LIN {X 0,Y 573.461,Z 507.991,A -85,B 0,C 180,E1 -2261.308,E2 -2261.308} C_VEL
LIN {X 0,Y 573.62,Z 497.143,A -85,B 0,C 180,E1 -2262.201,E2 -2262.201} C_VEL
LIN {X 0,Y 573.738,Z 485.26,A -85,B 0,C 180,E1 -2263.008,E2 -2263.008} C_VEL
LIN {X 0,Y 573.946,Z 472.1,A -85,B 0,C 180,E1 -2263.724,E2 -2263.724} C_VEL
LIN {X 0,Y 574.081,Z 458.765,A -85,B 0,C 180,E1 -2264.286,E2 -2264.286} C_VEL
LIN {X 0,Y 574.199,Z 444.491,A -85,B 0,C 180,E1 -2264.728,E2 -2264.728} C_VEL
LIN {X 0,Y 574.308,Z 429.641,A -85,B 0,C 180,E1 -2265.027,E2 -2265.027} C_VEL
LIN {X 0,Y 574.551,Z 299.634,A -85,B 0,C 180,E1 -2266.683,E2 -2266.683} C_VEL
LIN {X 0,Y 573.723,Z 294.688,A -85,B 0,C 180,E1 -2266.799,E2 -2266.799} C_VEL
LIN {X 0,Y 573.965,Z 271.516,A -85,B 0,C 180,E1 -2269.466,E2 -2269.466} C_VEL
LIN {X 0,Y 574.336,Z 247.477,A -85,B 0,C 180,E1 -2272.292,E2 -2272.292} C_VEL
LIN {X 0,Y 574.248,Z 241.135,A -85,B 0,C 180,E1 -2273.056,E2 -2273.056} C_VEL
LIN {X 0,Y 573.273,Z 236.765,A -85,B 0,C 180,E1 -2273.667,E2 -2273.667} C_VEL
LIN {X 0,Y 573.237,Z 236.705,A -85,B 0,C 180,E1 -2276.492,E2 -2276.492} C_VEL
LIN {X 0,Y 573.238,Z 236.705,A -85,B 0,C 180,E1 -2278.564,E2 -2278.564} C_VEL
LIN {X 0,Y 573.224,Z 236.702,A -85,B 0,C 180,E1 -2280.993,E2 -2280.993} C_VEL
LIN {X 0,Y 573.261,Z 236.697,A -85,B 0,C 180,E1 -2283.524,E2 -2283.524} C_VEL
LIN {X 0,Y 573.212,Z 236.706,A -85,B 0,C 180,E1 -2286.051,E2 -2286.051} C_VEL
LIN {X 0,Y 573.239,Z 236.705,A -85,B 0,C 180,E1 -2288.701,E2 -2288.701} C_VEL
LIN {X 0,Y 573.25,Z 236.698,A -85,B 0,C 180,E1 -2291.595,E2 -2291.595} C_VEL
LIN {X 0,Y 573.236,Z 236.707,A -85,B 0,C 180,E1 -2294.332,E2 -2294.332} C_VEL
LIN {X 0,Y 573.236,Z 236.7,A -85,B 0,C 180,E1 -2297.358,E2 -2297.358} C_VEL
LIN {X 0,Y 573.244,Z 236.706,A -85,B 0,C 180,E1 -2300.393,E2 -2300.393} C_VEL
LIN {X 0,Y 573.252,Z 236.696,A -85,B 0,C 180,E1 -2303.078,E2 -2303.078} C_VEL
LIN {X 0,Y 573.268,Z 236.698,A -85,B 0,C 180,E1 -2305.671,E2 -2305.671} C_VEL
LIN {X 0,Y 573.243,Z 236.705,A -85,B 0,C 180,E1 -2308.185,E2 -2308.185} C_VEL
LIN {X 0,Y 573.263,Z 236.695,A -85,B 0,C 180,E1 -2310.634,E2 -2310.634} C_VEL
LIN {X 0,Y 573.248,Z 236.698,A -85,B 0,C 180,E1 -2313.024,E2 -2313.024} C_VEL
LIN {X 0,Y 573.269,Z 236.697,A -85,B 0,C 180,E1 -2315.366,E2 -2315.366} C_VEL
LIN {X 0,Y 573.223,Z 236.703,A -85,B 0,C 180,E1 -2318.419,E2 -2318.419} C_VEL
LIN {X 0,Y 573.271,Z 236.695,A -85,B 0,C 180,E1 -2320.728,E2 -2320.728} C_VEL
LIN {X 0,Y 573.253,Z 236.704,A -85,B 0,C 180,E1 -2323.622,E2 -2323.622} C_VEL
LIN {X 0,Y 573.232,Z 236.7,A -85,B 0,C 180,E1 -2326.53,E2 -2326.53} C_VEL
LIN {X 0,Y 573.255,Z 236.696,A -85,B 0,C 180,E1 -2328.745,E2 -2328.745} C_VEL
LIN {X 0,Y 573.284,Z 236.701,A -85,B 0,C 180,E1 -2331.541,E2 -2331.541} C_VEL
LIN {X 0,Y 573.287,Z 236.694,A -85,B 0,C 180,E1 -2334.372,E2 -2334.372} C_VEL
LIN {X 0,Y 573.302,Z 236.696,A -85,B 0,C 180,E1 -2337.893,E2 -2337.893} C_VEL
LIN {X 0,Y 573.328,Z 236.688,A -85,B 0,C 180,E1 -2340.703,E2 -2340.703} C_VEL
LIN {X 0,Y 573.234,Z 236.71,A -85,B 0,C 180,E1 -2343.515,E2 -2343.515} C_VEL
LIN {X 0,Y 573.286,Z 236.7,A -85,B 0,C 180,E1 -2345.628,E2 -2345.628} C_VEL
LIN {X 0,Y 573.284,Z 236.693,A -85,B 0,C 180,E1 -2348.46,E2 -2348.46} C_VEL
LIN {X 0,Y 573.265,Z 236.705,A -85,B 0,C 180,E1 -2351.312,E2 -2351.312} C_VEL
LIN {X 0,Y 573.267,Z 236.696,A -85,B 0,C 180,E1 -2354.193,E2 -2354.193} C_VEL
LIN {X 0,Y 573.254,Z 236.704,A -85,B 0,C 180,E1 -2357.112,E2 -2357.112} C_VEL
LIN {X 0,Y 573.248,Z 236.697,A -85,B 0,C 180,E1 -2360.077,E2 -2360.077} C_VEL
LIN {X 0,Y 573.229,Z 236.71,A -85,B 0,C 180,E1 -2363.1,E2 -2363.1} C_VEL
LIN {X 0,Y 573.246,Z 236.698,A -85,B 0,C 180,E1 -2364.394,E2 -2364.394} C_VEL
LIN {X 0,Y 572.618,Z 236.785,A -85,B 0,C 180,E1 -2364.981,E2 -2364.981} C_VEL
LIN {X 0,Y 569.77,Z 237.14,A -85,B 0,C 180,E1 -2365.932,E2 -2365.932} C_VEL
LIN {X 0,Y 567.338,Z 237.443,A -85,B 0,C 180,E1 -2366.698,E2 -2366.698} C_VEL
LIN {X 0,Y 566.289,Z 237.57,A -85,B 0,C 180,E1 -2367.289,E2 -2367.289} C_VEL
LIN {X 0,Y 566.202,Z 237.577,A -85,B 0,C 180,E1 -2367.489,E2 -2367.489} C_VEL
LIN {X 0,Y 566.198,Z 237.575,A -85,B 0,C 180,E1 -2369.769,E2 -2369.769} C_VEL
LIN {X 0,Y 566.203,Z 237.578,A -85,B 0,C 180,E1 -2372.431,E2 -2372.431} C_VEL
LIN {X 0,Y 566.21,Z 237.581,A -85,B 0,C 180,E1 -2374.995,E2 -2374.995} C_VEL
LIN {X 0,Y 566.195,Z 237.579,A -85,B 0,C 180,E1 -2377.462,E2 -2377.462} C_VEL
LIN {X 0,Y 566.216,Z 237.572,A -85,B 0,C 180,E1 -2380.199,E2 -2380.199} C_VEL
LIN {X 0,Y 566.2,Z 237.581,A -85,B 0,C 180,E1 -2383.055,E2 -2383.055} C_VEL
LIN {X 0,Y 566.202,Z 237.577,A -85,B 0,C 180,E1 -2386.049,E2 -2386.049} C_VEL
LIN {X 0,Y 566.211,Z 237.583,A -85,B 0,C 180,E1 -2388.864,E2 -2388.864} C_VEL
LIN {X 0,Y 566.186,Z 237.572,A -85,B 0,C 180,E1 -2391.638,E2 -2391.638} C_VEL
LIN {X 0,Y 566.163,Z 237.586,A -85,B 0,C 180,E1 -2394.309,E2 -2394.309} C_VEL
LIN {X 0,Y 566.206,Z 237.583,A -85,B 0,C 180,E1 -2396.898,E2 -2396.898} C_VEL
LIN {X 0,Y 566.177,Z 237.58,A -85,B 0,C 180,E1 -2399.408,E2 -2399.408} C_VEL
LIN {X 0,Y 566.215,Z 237.575,A -85,B 0,C 180,E1 -2401.858,E2 -2401.858} C_VEL
LIN {X 0,Y 566.219,Z 237.771,A -85,B 0,C 180,E1 -2403.34,E2 -2403.34} C_VEL
LIN {X 0,Y 567.385,Z 244.16,A -85,B 0,C 180,E1 -2404.308,E2 -2404.308} C_VEL
LIN {X 0,Y 567.037,Z 265.173,A -85,B 0,C 180,E1 -2407.213,E2 -2407.213} C_VEL
LIN {X 0,Y 566.713,Z 286.13,A -85,B 0,C 180,E1 -2410.06,E2 -2410.06} C_VEL
LIN {X 0,Y 566.498,Z 307.4,A -85,B 0,C 180,E1 -2412.915,E2 -2412.915} C_VEL
LIN {X 0,Y 566.462,Z 315.728,A -85,B 0,C 180,E1 -2413.999,E2 -2413.999} C_VEL
LIN {X 0,Y 567.114,Z 320.48,A -85,B 0,C 180,E1 -2414.11,E2 -2414.11} C_VEL
LIN {X 0,Y 566.981,Z 424.267,A -85,B 0,C 180,E1 -2415.445,E2 -2415.445} C_VEL
LIN {X 0,Y 566.881,Z 437.515,A -85,B 0,C 180,E1 -2415.758,E2 -2415.758} C_VEL
LIN {X 0,Y 566.8,Z 449.793,A -85,B 0,C 180,E1 -2416.191,E2 -2416.191} C_VEL
LIN {X 0,Y 566.627,Z 461.317,A -85,B 0,C 180,E1 -2416.735,E2 -2416.735} C_VEL
LIN {X 0,Y 566.46,Z 473.127,A -85,B 0,C 180,E1 -2417.46,E2 -2417.46} C_VEL
LIN {X 0,Y 566.308,Z 483.69,A -85,B 0,C 180,E1 -2418.275,E2 -2418.275} C_VEL
LIN {X 0,Y 566.206,Z 492.834,A -85,B 0,C 180,E1 -2419.142,E2 -2419.142} C_VEL
LIN {X 0,Y 566.089,Z 501.649,A -85,B 0,C 180,E1 -2420.171,E2 -2420.171} C_VEL
LIN {X 0,Y 566.018,Z 509.117,A -85,B 0,C 180,E1 -2421.251,E2 -2421.251} C_VEL
LIN {X 0,Y 565.974,Z 515.994,A -85,B 0,C 180,E1 -2422.508,E2 -2422.508} C_VEL
LIN {X 0,Y 565.921,Z 520.519,A -85,B 0,C 180,E1 -2423.583,E2 -2423.583} C_VEL
LIN {X 0,Y 565.94,Z 522.904,A -85,B 0,C 180,E1 -2424.299,E2 -2424.299} C_VEL
LIN {X 0,Y 565.859,Z 524.856,A -85,B 0,C 180,E1 -2425.012,E2 -2425.012} C_VEL
LIN {X 0,Y 565.914,Z 526.392,A -85,B 0,C 180,E1 -2425.727,E2 -2425.727} C_VEL
LIN {X 0,Y 565.912,Z 527.482,A -85,B 0,C 180,E1 -2426.44,E2 -2426.44} C_VEL
LIN {X 0,Y 565.839,Z 528.467,A -85,B 0,C 180,E1 -2427.865,E2 -2427.865} C_VEL
LIN {X 0,Y 565.845,Z 528.388,A -85,B 0,C 180,E1 -2428.577,E2 -2428.577} C_VEL
LIN {X 0,Y 565.841,Z 527.885,A -85,B 0,C 180,E1 -2429.288,E2 -2429.288} C_VEL
LIN {X 0,Y 565.842,Z 526.984,A -85,B 0,C 180,E1 -2430,E2 -2430} C_VEL
LIN {X 0,Y 565.843,Z 525.687,A -85,B 0,C 180,E1 -2430.712,E2 -2430.712} C_VEL
LIN {X 0,Y 565.907,Z 522.941,A -85,B 0,C 180,E1 -2431.779,E2 -2431.779} C_VEL
LIN {X 0,Y 565.902,Z 519.185,A -85,B 0,C 180,E1 -2432.847,E2 -2432.847} C_VEL
LIN {X 0,Y 566.003,Z 514.319,A -85,B 0,C 180,E1 -2433.916,E2 -2433.916} C_VEL
LIN {X 0,Y 566.047,Z 508.196,A -85,B 0,C 180,E1 -2434.986,E2 -2434.986} C_VEL
LIN {X 0,Y 566.111,Z 500.59,A -85,B 0,C 180,E1 -2436.057,E2 -2436.057} C_VEL
LIN {X 0,Y 566.194,Z 492.807,A -85,B 0,C 180,E1 -2436.952,E2 -2436.952} C_VEL
LIN {X 0,Y 566.336,Z 482.261,A -85,B 0,C 180,E1 -2437.935,E2 -2437.935} C_VEL
LIN {X 0,Y 566.515,Z 471.518,A -85,B 0,C 180,E1 -2438.741,E2 -2438.741} C_VEL
LIN {X 0,Y 566.665,Z 461.053,A -85,B 0,C 180,E1 -2439.368,E2 -2439.368} C_VEL
LIN {X 0,Y 566.786,Z 449.616,A -85,B 0,C 180,E1 -2439.907,E2 -2439.907} C_VEL
LIN {X 0,Y 566.875,Z 436.702,A -85,B 0,C 180,E1 -2440.356,E2 -2440.356} C_VEL
LIN {X 0,Y 566.939,Z 424.14,A -85,B 0,C 180,E1 -2440.648,E2 -2440.648} C_VEL
LIN {X 0,Y 567.036,Z 319.865,A -85,B 0,C 180,E1 -2441.99,E2 -2441.99} C_VEL
LIN {X 0,Y 566.451,Z 315.894,A -85,B 0,C 180,E1 -2442.08,E2 -2442.08} C_VEL
LIN {X 0,Y 566.642,Z 298.504,A -85,B 0,C 180,E1 -2444.362,E2 -2444.362} C_VEL
LIN {X 0,Y 566.93,Z 274.221,A -85,B 0,C 180,E1 -2447.643,E2 -2447.643} C_VEL
LIN {X 0,Y 567.193,Z 253.473,A -85,B 0,C 180,E1 -2450.489,E2 -2450.489} C_VEL
LIN {X 0,Y 567.252,Z 242.568,A -85,B 0,C 180,E1 -2452.01,E2 -2452.01} C_VEL
LIN {X 0,Y 566.232,Z 237.708,A -85,B 0,C 180,E1 -2452.767,E2 -2452.767} C_VEL
LIN {X 0,Y 566.217,Z 237.569,A -85,B 0,C 180,E1 -2455.748,E2 -2455.748} C_VEL
LIN {X 0,Y 566.206,Z 237.578,A -85,B 0,C 180,E1 -2458.201,E2 -2458.201} C_VEL
LIN {X 0,Y 566.192,Z 237.581,A -85,B 0,C 180,E1 -2461.076,E2 -2461.076} C_VEL
LIN {X 0,Y 566.213,Z 237.577,A -85,B 0,C 180,E1 -2463.733,E2 -2463.733} C_VEL
LIN {X 0,Y 566.2,Z 237.578,A -85,B 0,C 180,E1 -2466.569,E2 -2466.569} C_VEL
LIN {X 0,Y 566.214,Z 237.578,A -85,B 0,C 180,E1 -2469.685,E2 -2469.685} C_VEL
LIN {X 0,Y 566.214,Z 237.575,A -85,B 0,C 180,E1 -2472.086,E2 -2472.086} C_VEL
LIN {X 0,Y 566.172,Z 237.586,A -85,B 0,C 180,E1 -2475.035,E2 -2475.035} C_VEL
LIN {X 0,Y 566.187,Z 237.579,A -85,B 0,C 180,E1 -2477.91,E2 -2477.91} C_VEL
LIN {X 0,Y 566.22,Z 237.574,A -85,B 0,C 180,E1 -2480.726,E2 -2480.726} C_VEL
LIN {X 0,Y 566.215,Z 237.575,A -85,B 0,C 180,E1 -2483.783,E2 -2483.783} C_VEL
LIN {X 0,Y 566.208,Z 237.572,A -85,B 0,C 180,E1 -2486.265,E2 -2486.265} C_VEL
LIN {X 0,Y 566.198,Z 237.584,A -85,B 0,C 180,E1 -2488.921,E2 -2488.921} C_VEL
LIN {X 0,Y 566.191,Z 237.585,A -85,B 0,C 180,E1 -2491.046,E2 -2491.046} C_VEL
LIN {X 0,Y 566.214,Z 237.577,A -85,B 0,C 180,E1 -2493.458,E2 -2493.458} C_VEL
LIN {X 0,Y 566.194,Z 237.575,A -85,B 0,C 180,E1 -2495.819,E2 -2495.819} C_VEL
LIN {X 0,Y 566.202,Z 237.584,A -85,B 0,C 180,E1 -2498.902,E2 -2498.902} C_VEL
LIN {X 0,Y 566.206,Z 237.579,A -85,B 0,C 180,E1 -2501.172,E2 -2501.172} C_VEL
LIN {X 0,Y 566.215,Z 237.575,A -85,B 0,C 180,E1 -2503.412,E2 -2503.412} C_VEL
LIN {X 0,Y 566.195,Z 237.58,A -85,B 0,C 180,E1 -2506.358,E2 -2506.358} C_VEL
LIN {X 0,Y 566.227,Z 237.581,A -85,B 0,C 180,E1 -2508.675,E2 -2508.675} C_VEL
LIN {X 0,Y 566.227,Z 237.573,A -85,B 0,C 180,E1 -2511.434,E2 -2511.434} C_VEL
LIN {X 0,Y 566.254,Z 237.575,A -85,B 0,C 180,E1 -2514.301,E2 -2514.301} C_VEL
LIN {X 0,Y 566.273,Z 237.568,A -85,B 0,C 180,E1 -2517.866,E2 -2517.866} C_VEL
LIN {X 0,Y 566.299,Z 237.568,A -85,B 0,C 180,E1 -2520.711,E2 -2520.711} C_VEL
LIN {X 0,Y 566.269,Z 237.571,A -85,B 0,C 180,E1 -2522.845,E2 -2522.845} C_VEL
LIN {X 0,Y 566.255,Z 237.569,A -85,B 0,C 180,E1 -2525.698,E2 -2525.698} C_VEL
LIN {X 0,Y 566.227,Z 237.579,A -85,B 0,C 180,E1 -2528.566,E2 -2528.566} C_VEL
LIN {X 0,Y 566.234,Z 237.571,A -85,B 0,C 180,E1 -2531.454,E2 -2531.454} C_VEL
LIN {X 0,Y 566.227,Z 237.577,A -85,B 0,C 180,E1 -2534.507,E2 -2534.507} C_VEL
LIN {X 0,Y 566.197,Z 237.576,A -85,B 0,C 180,E1 -2537.332,E2 -2537.332} C_VEL
LIN {X 0,Y 566.207,Z 237.581,A -85,B 0,C 180,E1 -2540.337,E2 -2540.337} C_VEL
LIN {X 0,Y 566.183,Z 237.579,A -85,B 0,C 180,E1 -2543.404,E2 -2543.404} C_VEL
LIN {X 0,Y 566.208,Z 237.579,A -85,B 0,C 180,E1 -2545.749,E2 -2545.749} C_VEL
LIN {X 0,Y 566.199,Z 237.581,A -85,B 0,C 180,E1 -2548.203,E2 -2548.203} C_VEL
LIN {X 0,Y 566.187,Z 237.576,A -85,B 0,C 180,E1 -2550.592,E2 -2550.592} C_VEL
LIN {X 0,Y 566.222,Z 237.574,A -85,B 0,C 180,E1 -2553.102,E2 -2553.102} C_VEL
LIN {X 0,Y 566.207,Z 237.582,A -85,B 0,C 180,E1 -2555.689,E2 -2555.689} C_VEL
LIN {X 0,Y 566.211,Z 237.576,A -85,B 0,C 180,E1 -2558.559,E2 -2558.559} C_VEL
LIN {X 0,Y 566.207,Z 237.576,A -85,B 0,C 180,E1 -2561.137,E2 -2561.137} C_VEL
LIN {X 0,Y 566.192,Z 237.583,A -85,B 0,C 180,E1 -2564.036,E2 -2564.036} C_VEL
LIN {X 0,Y 566.202,Z 237.574,A -85,B 0,C 180,E1 -2567.083,E2 -2567.083} C_VEL
LIN {X 0,Y 566.203,Z 237.583,A -85,B 0,C 180,E1 -2569.802,E2 -2569.802} C_VEL
LIN {X 0,Y 566.195,Z 237.576,A -85,B 0,C 180,E1 -2572.6,E2 -2572.6} C_VEL
LIN {X 0,Y 566.197,Z 237.577,A -85,B 0,C 180,E1 -2575.182,E2 -2575.182} C_VEL
LIN {X 0,Y 566.232,Z 237.575,A -85,B 0,C 180,E1 -2577.744,E2 -2577.744} C_VEL
LIN {X 0,Y 566.202,Z 237.577,A -85,B 0,C 180,E1 -2580.328,E2 -2580.328} C_VEL
LIN {X 0,Y 566.211,Z 237.578,A -85,B 0,C 180,E1 -2582.661,E2 -2582.661} C_VEL
LIN {X 0,Y 566.236,Z 237.579,A -85,B 0,C 180,E1 -2585.04,E2 -2585.04} C_VEL
LIN {X 0,Y 566.236,Z 237.751,A -85,B 0,C 180,E1 -2586.162,E2 -2586.162} C_VEL
LIN {X 0,Y 567.57,Z 244.334,A -85,B 0,C 180,E1 -2587.043,E2 -2587.043} C_VEL
LIN {X 0,Y 567.133,Z 270.032,A -85,B 0,C 180,E1 -2590.114,E2 -2590.114} C_VEL
LIN {X 0,Y 566.764,Z 294.641,A -85,B 0,C 180,E1 -2592.989,E2 -2592.989} C_VEL
LIN {X 0,Y 567.781,Z 300.586,A -85,B 0,C 180,E1 -2593.125,E2 -2593.125} C_VEL
LIN {X 0,Y 567.463,Z 432.653,A -85,B 0,C 180,E1 -2594.833,E2 -2594.833} C_VEL
LIN {X 0,Y 567.338,Z 447.003,A -85,B 0,C 180,E1 -2595.156,E2 -2595.156} C_VEL
LIN {X 0,Y 567.188,Z 460.402,A -85,B 0,C 180,E1 -2595.599,E2 -2595.599} C_VEL
LIN {X 0,Y 567.011,Z 473.882,A -85,B 0,C 180,E1 -2596.196,E2 -2596.196} C_VEL
LIN {X 0,Y 566.77,Z 486.682,A -85,B 0,C 180,E1 -2596.921,E2 -2596.921} C_VEL
LIN {X 0,Y 566.615,Z 498.315,A -85,B 0,C 180,E1 -2597.737,E2 -2597.737} C_VEL
LIN {X 0,Y 566.443,Z 508.223,A -85,B 0,C 180,E1 -2598.572,E2 -2598.572} C_VEL
LIN {X 0,Y 566.294,Z 518.709,A -85,B 0,C 180,E1 -2599.633,E2 -2599.633} C_VEL
LIN {X 0,Y 566.18,Z 527.559,A -85,B 0,C 180,E1 -2600.714,E2 -2600.714} C_VEL
LIN {X 0,Y 566.047,Z 536.037,A -85,B 0,C 180,E1 -2601.971,E2 -2601.971} C_VEL
LIN {X 0,Y 565.966,Z 543.803,A -85,B 0,C 180,E1 -2603.422,E2 -2603.422} C_VEL
LIN {X 0,Y 565.928,Z 548.961,A -85,B 0,C 180,E1 -2604.656,E2 -2604.656} C_VEL
LIN {X 0,Y 565.956,Z 552.444,A -85,B 0,C 180,E1 -2605.727,E2 -2605.727} C_VEL
LIN {X 0,Y 565.875,Z 555.832,A -85,B 0,C 180,E1 -2607.153,E2 -2607.153} C_VEL
LIN {X 0,Y 565.841,Z 557.833,A -85,B 0,C 180,E1 -2608.577,E2 -2608.577} C_VEL
LIN {X 0,Y 565.837,Z 558.5,A -85,B 0,C 180,E1 -2610,E2 -2610} C_VEL
LIN {X 0,Y 565.841,Z 557.834,A -85,B 0,C 180,E1 -2611.423,E2 -2611.423} C_VEL
LIN {X 0,Y 565.875,Z 555.834,A -85,B 0,C 180,E1 -2612.848,E2 -2612.848} C_VEL
LIN {X 0,Y 565.956,Z 552.446,A -85,B 0,C 180,E1 -2614.273,E2 -2614.273} C_VEL
LIN {X 0,Y 565.985,Z 547.568,A -85,B 0,C 180,E1 -2615.701,E2 -2615.701} C_VEL
LIN {X 0,Y 565.995,Z 543.044,A -85,B 0,C 180,E1 -2616.739,E2 -2616.739} C_VEL
LIN {X 0,Y 566.047,Z 536.037,A -85,B 0,C 180,E1 -2618.029,E2 -2618.029} C_VEL
LIN {X 0,Y 566.177,Z 527.558,A -85,B 0,C 180,E1 -2619.286,E2 -2619.286} C_VEL
LIN {X 0,Y 566.294,Z 518.708,A -85,B 0,C 180,E1 -2620.367,E2 -2620.367} C_VEL
LIN {X 0,Y 566.485,Z 507.99,A -85,B 0,C 180,E1 -2621.449,E2 -2621.449} C_VEL
LIN {X 0,Y 566.611,Z 497.14,A -85,B 0,C 180,E1 -2622.354,E2 -2622.354} C_VEL
LIN {X 0,Y 566.778,Z 485.257,A -85,B 0,C 180,E1 -2623.17,E2 -2623.17} C_VEL
LIN {X 0,Y 567.033,Z 472.1,A -85,B 0,C 180,E1 -2623.895,E2 -2623.895} C_VEL
LIN {X 0,Y 567.212,Z 458.959,A -85,B 0,C 180,E1 -2624.456,E2 -2624.456} C_VEL
LIN {X 0,Y 567.323,Z 444.842,A -85,B 0,C 180,E1 -2624.902,E2 -2624.902} C_VEL
LIN {X 0,Y 567.457,Z 431.144,A -85,B 0,C 180,E1 -2625.19,E2 -2625.19} C_VEL
LIN {X 0,Y 567.777,Z 300.723,A -85,B 0,C 180,E1 -2626.873,E2 -2626.873} C_VEL
LIN {X 0,Y 566.792,Z 294.745,A -85,B 0,C 180,E1 -2627.007,E2 -2627.007} C_VEL
LIN {X 0,Y 567.091,Z 271.462,A -85,B 0,C 180,E1 -2629.718,E2 -2629.718} C_VEL
LIN {X 0,Y 567.538,Z 245.923,A -85,B 0,C 180,E1 -2632.766,E2 -2632.766} C_VEL
LIN {X 0,Y 567.04,Z 241.168,A -85,B 0,C 180,E1 -2633.366,E2 -2633.366} C_VEL
LIN {X 0,Y 566.214,Z 237.67,A -85,B 0,C 180,E1 -2633.863,E2 -2633.863} C_VEL
LIN {X 0,Y 566.208,Z 237.582,A -85,B 0,C 180,E1 -2636.659,E2 -2636.659} C_VEL
LIN {X 0,Y 566.192,Z 237.581,A -85,B 0,C 180,E1 -2638.953,E2 -2638.953} C_VEL
LIN {X 0,Y 566.192,Z 237.576,A -85,B 0,C 180,E1 -2641.421,E2 -2641.421} C_VEL
LIN {X 0,Y 566.208,Z 237.578,A -85,B 0,C 180,E1 -2643.955,E2 -2643.955} C_VEL
LIN {X 0,Y 566.197,Z 237.58,A -85,B 0,C 180,E1 -2646.569,E2 -2646.569} C_VEL
LIN {X 0,Y 566.213,Z 237.576,A -85,B 0,C 180,E1 -2649.685,E2 -2649.685} C_VEL
LIN {X 0,Y 566.211,Z 237.58,A -85,B 0,C 180,E1 -2652.087,E2 -2652.087} C_VEL
LIN {X 0,Y 566.17,Z 237.58,A -85,B 0,C 180,E1 -2655.035,E2 -2655.035} C_VEL
LIN {X 0,Y 566.213,Z 237.582,A -85,B 0,C 180,E1 -2658.135,E2 -2658.135} C_VEL
LIN {X 0,Y 566.218,Z 237.576,A -85,B 0,C 180,E1 -2660.727,E2 -2660.727} C_VEL
LIN {X 0,Y 566.213,Z 237.577,A -85,B 0,C 180,E1 -2663.783,E2 -2663.783} C_VEL
LIN {X 0,Y 566.207,Z 237.583,A -85,B 0,C 180,E1 -2666.265,E2 -2666.265} C_VEL
LIN {X 0,Y 566.196,Z 237.575,A -85,B 0,C 180,E1 -2668.921,E2 -2668.921} C_VEL
LIN {X 0,Y 566.189,Z 237.575,A -85,B 0,C 180,E1 -2671.047,E2 -2671.047} C_VEL
LIN {X 0,Y 566.212,Z 237.577,A -85,B 0,C 180,E1 -2673.459,E2 -2673.459} C_VEL
LIN {X 0,Y 566.194,Z 237.585,A -85,B 0,C 180,E1 -2675.819,E2 -2675.819} C_VEL
LIN {X 0,Y 566.201,Z 237.575,A -85,B 0,C 180,E1 -2678.902,E2 -2678.902} C_VEL
LIN {X 0,Y 566.206,Z 237.576,A -85,B 0,C 180,E1 -2681.172,E2 -2681.172} C_VEL
LIN {X 0,Y 566.214,Z 237.578,A -85,B 0,C 180,E1 -2683.413,E2 -2683.413} C_VEL
LIN {X 0,Y 566.194,Z 237.578,A -85,B 0,C 180,E1 -2686.359,E2 -2686.359} C_VEL
LIN {X 0,Y 566.227,Z 237.572,A -85,B 0,C 180,E1 -2688.675,E2 -2688.675} C_VEL
LIN {X 0,Y 566.228,Z 237.579,A -85,B 0,C 180,E1 -2691.434,E2 -2691.434} C_VEL
LIN {X 0,Y 566.255,Z 237.57,A -85,B 0,C 180,E1 -2694.302,E2 -2694.302} C_VEL
LIN {X 0,Y 566.273,Z 237.572,A -85,B 0,C 180,E1 -2697.866,E2 -2697.866} C_VEL
LIN {X 0,Y 566.298,Z 237.564,A -85,B 0,C 180,E1 -2700.711,E2 -2700.711} C_VEL
LIN {X 0,Y 566.27,Z 237.567,A -85,B 0,C 180,E1 -2702.846,E2 -2702.846} C_VEL
LIN {X 0,Y 566.254,Z 237.574,A -85,B 0,C 180,E1 -2705.699,E2 -2705.699} C_VEL
LIN {X 0,Y 566.228,Z 237.573,A -85,B 0,C 180,E1 -2708.566,E2 -2708.566} C_VEL
LIN {X 0,Y 566.235,Z 237.58,A -85,B 0,C 180,E1 -2711.455,E2 -2711.455} C_VEL
LIN {X 0,Y 566.228,Z 237.573,A -85,B 0,C 180,E1 -2714.507,E2 -2714.507} C_VEL
LIN {X 0,Y 566.199,Z 237.585,A -85,B 0,C 180,E1 -2717.332,E2 -2717.332} C_VEL
LIN {X 0,Y 566.209,Z 237.574,A -85,B 0,C 180,E1 -2720.338,E2 -2720.338} C_VEL
LIN {X 0,Y 566.185,Z 237.583,A -85,B 0,C 180,E1 -2723.404,E2 -2723.404} C_VEL
LIN {X 0,Y 566.21,Z 237.577,A -85,B 0,C 180,E1 -2725.75,E2 -2725.75} C_VEL
LIN {X 0,Y 566.202,Z 237.577,A -85,B 0,C 180,E1 -2727.489,E2 -2727.489} C_VEL
LIN {X 0,Y 565.53,Z 237.659,A -85,B 0,C 180,E1 -2728.083,E2 -2728.083} C_VEL
LIN {X 0,Y 562.664,Z 238.021,A -85,B 0,C 180,E1 -2729.046,E2 -2729.046} C_VEL
LIN {X 0,Y 560.249,Z 238.318,A -85,B 0,C 180,E1 -2729.822,E2 -2729.822} C_VEL
LIN {X 0,Y 559.221,Z 238.445,A -85,B 0,C 180,E1 -2730.421,E2 -2730.421} C_VEL
LIN {X 0,Y 559.142,Z 238.457,A -85,B 0,C 180,E1 -2730.623,E2 -2730.623} C_VEL
LIN {X 0,Y 559.162,Z 238.453,A -85,B 0,C 180,E1 -2733.575,E2 -2733.575} C_VEL
LIN {X 0,Y 559.167,Z 238.453,A -85,B 0,C 180,E1 -2736.449,E2 -2736.449} C_VEL
LIN {X 0,Y 559.177,Z 238.458,A -85,B 0,C 180,E1 -2738.934,E2 -2738.934} C_VEL
LIN {X 0,Y 559.164,Z 238.453,A -85,B 0,C 180,E1 -2741.771,E2 -2741.771} C_VEL
LIN {X 0,Y 559.139,Z 238.462,A -85,B 0,C 180,E1 -2744.74,E2 -2744.74} C_VEL
LIN {X 0,Y 559.164,Z 238.454,A -85,B 0,C 180,E1 -2747.258,E2 -2747.258} C_VEL
LIN {X 0,Y 559.18,Z 238.453,A -85,B 0,C 180,E1 -2750.135,E2 -2750.135} C_VEL
LIN {X 0,Y 559.142,Z 238.463,A -85,B 0,C 180,E1 -2752.892,E2 -2752.892} C_VEL
LIN {X 0,Y 559.157,Z 238.453,A -85,B 0,C 180,E1 -2756.053,E2 -2756.053} C_VEL
LIN {X 0,Y 559.155,Z 238.456,A -85,B 0,C 180,E1 -2758.981,E2 -2758.981} C_VEL
LIN {X 0,Y 559.148,Z 238.454,A -85,B 0,C 180,E1 -2761.624,E2 -2761.624} C_VEL
LIN {X 0,Y 559.196,Z 238.639,A -85,B 0,C 180,E1 -2763.141,E2 -2763.141} C_VEL
LIN {X 0,Y 560.458,Z 245.124,A -85,B 0,C 180,E1 -2764.14,E2 -2764.14} C_VEL
LIN {X 0,Y 560.166,Z 264.949,A -85,B 0,C 180,E1 -2766.917,E2 -2766.917} C_VEL
LIN {X 0,Y 559.762,Z 285.913,A -85,B 0,C 180,E1 -2769.802,E2 -2769.802} C_VEL
LIN {X 0,Y 559.517,Z 307.055,A -85,B 0,C 180,E1 -2772.675,E2 -2772.675} C_VEL
LIN {X 0,Y 559.446,Z 315.449,A -85,B 0,C 180,E1 -2773.792,E2 -2773.792} C_VEL
LIN {X 0,Y 559.889,Z 319.091,A -85,B 0,C 180,E1 -2773.908,E2 -2773.908} C_VEL
LIN {X 0,Y 560.332,Z 321.906,A -85,B 0,C 180,E1 -2773.956,E2 -2773.956} C_VEL
LIN {X 0,Y 560.072,Z 424.516,A -85,B 0,C 180,E1 -2775.292,E2 -2775.292} C_VEL
LIN {X 0,Y 559.961,Z 437.437,A -85,B 0,C 180,E1 -2775.602,E2 -2775.602} C_VEL
LIN {X 0,Y 559.852,Z 450.302,A -85,B 0,C 180,E1 -2776.063,E2 -2776.063} C_VEL
LIN {X 0,Y 559.628,Z 462.495,A -85,B 0,C 180,E1 -2776.658,E2 -2776.658} C_VEL
LIN {X 0,Y 559.454,Z 474.066,A -85,B 0,C 180,E1 -2777.393,E2 -2777.393} C_VEL
LIN {X 0,Y 559.268,Z 484.463,A -85,B 0,C 180,E1 -2778.217,E2 -2778.217} C_VEL
LIN {X 0,Y 559.14,Z 493.794,A -85,B 0,C 180,E1 -2779.133,E2 -2779.133} C_VEL
LIN {X 0,Y 559.008,Z 502.821,A -85,B 0,C 180,E1 -2780.228,E2 -2780.228} C_VEL
LIN {X 0,Y 558.933,Z 510.083,A -85,B 0,C 180,E1 -2781.322,E2 -2781.322} C_VEL
LIN {X 0,Y 558.899,Z 515.879,A -85,B 0,C 180,E1 -2782.413,E2 -2782.413} C_VEL
LIN {X 0,Y 558.819,Z 521.124,A -85,B 0,C 180,E1 -2783.702,E2 -2783.702} C_VEL
LIN {X 0,Y 558.775,Z 524.795,A -85,B 0,C 180,E1 -2784.949,E2 -2784.949} C_VEL
LIN {X 0,Y 558.807,Z 526.343,A -85,B 0,C 180,E1 -2785.672,E2 -2785.672} C_VEL
LIN {X 0,Y 558.821,Z 527.454,A -85,B 0,C 180,E1 -2786.395,E2 -2786.395} C_VEL
LIN {X 0,Y 558.745,Z 528.461,A -85,B 0,C 180,E1 -2787.837,E2 -2787.837} C_VEL
LIN {X 0,Y 558.745,Z 528.394,A -85,B 0,C 180,E1 -2788.558,E2 -2788.558} C_VEL
LIN {X 0,Y 558.741,Z 527.913,A -85,B 0,C 180,E1 -2789.279,E2 -2789.279} C_VEL
LIN {X 0,Y 558.744,Z 525.737,A -85,B 0,C 180,E1 -2790.721,E2 -2790.721} C_VEL
LIN {X 0,Y 558.823,Z 523.014,A -85,B 0,C 180,E1 -2791.802,E2 -2791.802} C_VEL
LIN {X 0,Y 558.826,Z 519.283,A -85,B 0,C 180,E1 -2792.883,E2 -2792.883} C_VEL
LIN {X 0,Y 558.908,Z 514.444,A -85,B 0,C 180,E1 -2793.966,E2 -2793.966} C_VEL
LIN {X 0,Y 558.972,Z 508.35,A -85,B 0,C 180,E1 -2795.049,E2 -2795.049} C_VEL
LIN {X 0,Y 559.07,Z 500.783,A -85,B 0,C 180,E1 -2796.134,E2 -2796.134} C_VEL
LIN {X 0,Y 559.163,Z 492.315,A -85,B 0,C 180,E1 -2797.115,E2 -2797.115} C_VEL
LIN {X 0,Y 559.328,Z 482.554,A -85,B 0,C 180,E1 -2798.035,E2 -2798.035} C_VEL
LIN {X 0,Y 559.517,Z 471.874,A -85,B 0,C 180,E1 -2798.851,E2 -2798.851} C_VEL
LIN {X 0,Y 559.694,Z 461.519,A -85,B 0,C 180,E1 -2799.486,E2 -2799.486} C_VEL
LIN {X 0,Y 559.81,Z 450.236,A -85,B 0,C 180,E1 -2800.031,E2 -2800.031} C_VEL
LIN {X 0,Y 559.93,Z 436.781,A -85,B 0,C 180,E1 -2800.509,E2 -2800.509} C_VEL
LIN {X 0,Y 560.031,Z 424.26,A -85,B 0,C 180,E1 -2800.804,E2 -2800.804} C_VEL
LIN {X 0,Y 560.247,Z 321.307,A -85,B 0,C 180,E1 -2802.144,E2 -2802.144} C_VEL
LIN {X 0,Y 559.524,Z 316.503,A -85,B 0,C 180,E1 -2802.251,E2 -2802.251} C_VEL
LIN {X 0,Y 559.409,Z 315.105,A -85,B 0,C 180,E1 -2802.332,E2 -2802.332} C_VEL
LIN {X 0,Y 559.701,Z 294.577,A -85,B 0,C 180,E1 -2805.106,E2 -2805.106} C_VEL
LIN {X 0,Y 560.034,Z 272.757,A -85,B 0,C 180,E1 -2808.095,E2 -2808.095} C_VEL
LIN {X 0,Y 560.349,Z 252.275,A -85,B 0,C 180,E1 -2810.943,E2 -2810.943} C_VEL
LIN {X 0,Y 560.347,Z 244.092,A -85,B 0,C 180,E1 -2812.102,E2 -2812.102} C_VEL
LIN {X 0,Y 559.184,Z 238.577,A -85,B 0,C 180,E1 -2812.966,E2 -2812.966} C_VEL
LIN {X 0,Y 559.182,Z 238.448,A -85,B 0,C 180,E1 -2816.096,E2 -2816.096} C_VEL
LIN {X 0,Y 559.166,Z 238.454,A -85,B 0,C 180,E1 -2818.529,E2 -2818.529} C_VEL
LIN {X 0,Y 559.148,Z 238.461,A -85,B 0,C 180,E1 -2821.272,E2 -2821.272} C_VEL
LIN {X 0,Y 559.167,Z 238.452,A -85,B 0,C 180,E1 -2823.948,E2 -2823.948} C_VEL
LIN {X 0,Y 559.141,Z 238.463,A -85,B 0,C 180,E1 -2827.108,E2 -2827.108} C_VEL
LIN {X 0,Y 559.16,Z 238.454,A -85,B 0,C 180,E1 -2829.941,E2 -2829.941} C_VEL
LIN {X 0,Y 559.164,Z 238.455,A -85,B 0,C 180,E1 -2832.742,E2 -2832.742} C_VEL
LIN {X 0,Y 559.151,Z 238.455,A -85,B 0,C 180,E1 -2835.76,E2 -2835.76} C_VEL
LIN {X 0,Y 559.163,Z 238.453,A -85,B 0,C 180,E1 -2838.229,E2 -2838.229} C_VEL
LIN {X 0,Y 559.176,Z 238.459,A -85,B 0,C 180,E1 -2841.19,E2 -2841.19} C_VEL
LIN {X 0,Y 559.17,Z 238.452,A -85,B 0,C 180,E1 -2843.791,E2 -2843.791} C_VEL
LIN {X 0,Y 559.161,Z 238.45,A -85,B 0,C 180,E1 -2846.425,E2 -2846.425} C_VEL
LIN {X 0,Y 559.162,Z 238.462,A -85,B 0,C 180,E1 -2848.981,E2 -2848.981} C_VEL
LIN {X 0,Y 559.163,Z 238.453,A -85,B 0,C 180,E1 -2851.618,E2 -2851.618} C_VEL
LIN {X 0,Y 559.177,Z 238.451,A -85,B 0,C 180,E1 -2853.902,E2 -2853.902} C_VEL
LIN {X 0,Y 559.151,Z 238.458,A -85,B 0,C 180,E1 -2856.567,E2 -2856.567} C_VEL
LIN {X 0,Y 559.174,Z 238.452,A -85,B 0,C 180,E1 -2859.395,E2 -2859.395} C_VEL
LIN {X 0,Y 559.148,Z 238.455,A -85,B 0,C 180,E1 -2861.685,E2 -2861.685} C_VEL
LIN {X 0,Y 559.164,Z 238.453,A -85,B 0,C 180,E1 -2863.947,E2 -2863.947} C_VEL
LIN {X 0,Y 559.168,Z 238.453,A -85,B 0,C 180,E1 -2866.184,E2 -2866.184} C_VEL
LIN {X 0,Y 559.188,Z 238.451,A -85,B 0,C 180,E1 -2869.133,E2 -2869.133} C_VEL
LIN {X 0,Y 559.2,Z 238.45,A -85,B 0,C 180,E1 -2872.053,E2 -2872.053} C_VEL
LIN {X 0,Y 559.25,Z 238.443,A -85,B 0,C 180,E1 -2874.953,E2 -2874.953} C_VEL
LIN {X 0,Y 559.245,Z 238.444,A -85,B 0,C 180,E1 -2877.839,E2 -2877.839} C_VEL
LIN {X 0,Y 559.269,Z 238.444,A -85,B 0,C 180,E1 -2880.72,E2 -2880.72} C_VEL
LIN {X 0,Y 559.235,Z 238.447,A -85,B 0,C 180,E1 -2882.881,E2 -2882.881} C_VEL
LIN {X 0,Y 559.224,Z 238.445,A -85,B 0,C 180,E1 -2885.77,E2 -2885.77} C_VEL
LIN {X 0,Y 559.186,Z 238.454,A -85,B 0,C 180,E1 -2888.674,E2 -2888.674} C_VEL
LIN {X 0,Y 559.197,Z 238.448,A -85,B 0,C 180,E1 -2891.6,E2 -2891.6} C_VEL
LIN {X 0,Y 559.192,Z 238.452,A -85,B 0,C 180,E1 -2894.596,E2 -2894.596} C_VEL
LIN {X 0,Y 559.156,Z 238.455,A -85,B 0,C 180,E1 -2897.557,E2 -2897.557} C_VEL
LIN {X 0,Y 559.165,Z 238.457,A -85,B 0,C 180,E1 -2899.837,E2 -2899.837} C_VEL
LIN {X 0,Y 559.135,Z 238.466,A -85,B 0,C 180,E1 -2902.153,E2 -2902.153} C_VEL
LIN {X 0,Y 559.172,Z 238.451,A -85,B 0,C 180,E1 -2905.187,E2 -2905.187} C_VEL
LIN {X 0,Y 559.186,Z 238.455,A -85,B 0,C 180,E1 -2907.712,E2 -2907.712} C_VEL
LIN {X 0,Y 559.162,Z 238.456,A -85,B 0,C 180,E1 -2910.182,E2 -2910.182} C_VEL
LIN {X 0,Y 559.169,Z 238.453,A -85,B 0,C 180,E1 -2912.714,E2 -2912.714} C_VEL
LIN {X 0,Y 559.153,Z 238.456,A -85,B 0,C 180,E1 -2915.322,E2 -2915.322} C_VEL
LIN {X 0,Y 559.13,Z 238.464,A -85,B 0,C 180,E1 -2918.018,E2 -2918.018} C_VEL
LIN {X 0,Y 559.172,Z 238.452,A -85,B 0,C 180,E1 -2920.811,E2 -2920.811} C_VEL
LIN {X 0,Y 559.155,Z 238.462,A -85,B 0,C 180,E1 -2923.733,E2 -2923.733} C_VEL
LIN {X 0,Y 559.146,Z 238.451,A -85,B 0,C 180,E1 -2926.803,E2 -2926.803} C_VEL
LIN {X 0,Y 559.155,Z 238.45,A -85,B 0,C 180,E1 -2929.188,E2 -2929.188} C_VEL
LIN {X 0,Y 559.13,Z 238.461,A -85,B 0,C 180,E1 -2931.983,E2 -2931.983} C_VEL
LIN {X 0,Y 559.13,Z 238.454,A -85,B 0,C 180,E1 -2934.788,E2 -2934.788} C_VEL
LIN {X 0,Y 559.173,Z 238.46,A -85,B 0,C 180,E1 -2937.362,E2 -2937.362} C_VEL
LIN {X 0,Y 559.147,Z 238.457,A -85,B 0,C 180,E1 -2940.143,E2 -2940.143} C_VEL
LIN {X 0,Y 559.169,Z 238.459,A -85,B 0,C 180,E1 -2943.098,E2 -2943.098} C_VEL
LIN {X 0,Y 559.195,Z 238.597,A -85,B 0,C 180,E1 -2945.942,E2 -2945.942} C_VEL
LIN {X 0,Y 560.726,Z 246.098,A -85,B 0,C 180,E1 -2946.96,E2 -2946.96} C_VEL
LIN {X 0,Y 560.227,Z 271.286,A -85,B 0,C 180,E1 -2950.011,E2 -2950.011} C_VEL
LIN {X 0,Y 559.841,Z 294.817,A -85,B 0,C 180,E1 -2952.784,E2 -2952.784} C_VEL
LIN {X 0,Y 561.014,Z 302.282,A -85,B 0,C 180,E1 -2952.937,E2 -2952.937} C_VEL
LIN {X 0,Y 560.615,Z 432.653,A -85,B 0,C 180,E1 -2954.644,E2 -2954.644} C_VEL
LIN {X 0,Y 560.47,Z 446.942,A -85,B 0,C 180,E1 -2954.968,E2 -2954.968} C_VEL
LIN {X 0,Y 560.307,Z 460.487,A -85,B 0,C 180,E1 -2955.421,E2 -2955.421} C_VEL
LIN {X 0,Y 560.105,Z 473.88,A -85,B 0,C 180,E1 -2956.023,E2 -2956.023} C_VEL
LIN {X 0,Y 559.81,Z 486.679,A -85,B 0,C 180,E1 -2956.755,E2 -2956.755} C_VEL
LIN {X 0,Y 559.635,Z 498.313,A -85,B 0,C 180,E1 -2957.581,E2 -2957.581} C_VEL
LIN {X 0,Y 559.43,Z 508.919,A -85,B 0,C 180,E1 -2958.492,E2 -2958.492} C_VEL
LIN {X 0,Y 559.272,Z 518.709,A -85,B 0,C 180,E1 -2959.502,E2 -2959.502} C_VEL
LIN {X 0,Y 559.121,Z 527.559,A -85,B 0,C 180,E1 -2960.596,E2 -2960.596} C_VEL
LIN {X 0,Y 558.986,Z 536.036,A -85,B 0,C 180,E1 -2961.869,E2 -2961.869} C_VEL
LIN {X 0,Y 558.901,Z 542.866,A -85,B 0,C 180,E1 -2963.14,E2 -2963.14} C_VEL
LIN {X 0,Y 558.913,Z 547.569,A -85,B 0,C 180,E1 -2964.227,E2 -2964.227} C_VEL
LIN {X 0,Y 558.865,Z 552.444,A -85,B 0,C 180,E1 -2965.673,E2 -2965.673} C_VEL
LIN {X 0,Y 558.796,Z 555.832,A -85,B 0,C 180,E1 -2967.116,E2 -2967.116} C_VEL
LIN {X 0,Y 558.74,Z 557.834,A -85,B 0,C 180,E1 -2968.559,E2 -2968.559} C_VEL
LIN {X 0,Y 558.738,Z 558.5,A -85,B 0,C 180,E1 -2970,E2 -2970} C_VEL
LIN {X 0,Y 558.74,Z 557.835,A -85,B 0,C 180,E1 -2971.442,E2 -2971.442} C_VEL
LIN {X 0,Y 558.796,Z 555.835,A -85,B 0,C 180,E1 -2972.884,E2 -2972.884} C_VEL
LIN {X 0,Y 558.865,Z 552.446,A -85,B 0,C 180,E1 -2974.327,E2 -2974.327} C_VEL
LIN {X 0,Y 558.914,Z 547.568,A -85,B 0,C 180,E1 -2975.773,E2 -2975.773} C_VEL
LIN {X 0,Y 558.906,Z 541.054,A -85,B 0,C 180,E1 -2977.224,E2 -2977.224} C_VEL
LIN {X 0,Y 559.028,Z 533.803,A -85,B 0,C 180,E1 -2978.495,E2 -2978.495} C_VEL
LIN {X 0,Y 559.146,Z 524.823,A -85,B 0,C 180,E1 -2979.769,E2 -2979.769} C_VEL
LIN {X 0,Y 559.35,Z 515.394,A -85,B 0,C 180,E1 -2980.863,E2 -2980.863} C_VEL
LIN {X 0,Y 559.518,Z 504.956,A -85,B 0,C 180,E1 -2981.869,E2 -2981.869} C_VEL
LIN {X 0,Y 559.708,Z 493.433,A -85,B 0,C 180,E1 -2982.786,E2 -2982.786} C_VEL
LIN {X 0,Y 559.923,Z 480.643,A -85,B 0,C 180,E1 -2983.612,E2 -2983.612} C_VEL
LIN {X 0,Y 560.165,Z 468.152,A -85,B 0,C 180,E1 -2984.254,E2 -2984.254} C_VEL
LIN {X 0,Y 560.404,Z 454.317,A -85,B 0,C 180,E1 -2984.802,E2 -2984.802} C_VEL
LIN {X 0,Y 560.55,Z 440.68,A -85,B 0,C 180,E1 -2985.192,E2 -2985.192} C_VEL
LIN {X 0,Y 560.624,Z 426.618,A -85,B 0,C 180,E1 -2985.449,E2 -2985.449} C_VEL
LIN {X 0,Y 560.942,Z 301.286,A -85,B 0,C 180,E1 -2987.078,E2 -2987.078} C_VEL
LIN {X 0,Y 559.846,Z 294.754,A -85,B 0,C 180,E1 -2987.225,E2 -2987.225} C_VEL
LIN {X 0,Y 560.22,Z 271.286,A -85,B 0,C 180,E1 -2989.989,E2 -2989.989} C_VEL
LIN {X 0,Y 560.717,Z 246.099,A -85,B 0,C 180,E1 -2993.041,E2 -2993.041} C_VEL
LIN {X 0,Y 559.17,Z 238.528,A -85,B 0,C 180,E1 -2994.084,E2 -2994.084} C_VEL
LIN {X 0,Y 559.169,Z 238.459,A -85,B 0,C 180,E1 -2996.902,E2 -2996.902} C_VEL
LIN {X 0,Y 559.147,Z 238.457,A -85,B 0,C 180,E1 -2999.857,E2 -2999.857} C_VEL
LIN {X 0,Y 559.174,Z 238.458,A -85,B 0,C 180,E1 -3002.713,E2 -3002.713} C_VEL
LIN {X 0,Y 559.126,Z 238.456,A -85,B 0,C 180,E1 -3005.324,E2 -3005.324} C_VEL
LIN {X 0,Y 559.13,Z 238.458,A -85,B 0,C 180,E1 -3008.017,E2 -3008.017} C_VEL
LIN {X 0,Y 559.156,Z 238.456,A -85,B 0,C 180,E1 -3010.812,E2 -3010.812} C_VEL
LIN {X 0,Y 559.16,Z 238.455,A -85,B 0,C 180,E1 -3013.731,E2 -3013.731} C_VEL
LIN {X 0,Y 559.142,Z 238.458,A -85,B 0,C 180,E1 -3016.803,E2 -3016.803} C_VEL
LIN {X 0,Y 559.172,Z 238.449,A -85,B 0,C 180,E1 -3019.189,E2 -3019.189} C_VEL
LIN {X 0,Y 559.13,Z 238.464,A -85,B 0,C 180,E1 -3021.982,E2 -3021.982} C_VEL
LIN {X 0,Y 559.154,Z 238.453,A -85,B 0,C 180,E1 -3024.783,E2 -3024.783} C_VEL
LIN {X 0,Y 559.168,Z 238.453,A -85,B 0,C 180,E1 -3027.361,E2 -3027.361} C_VEL
LIN {X 0,Y 559.183,Z 238.454,A -85,B 0,C 180,E1 -3030.135,E2 -3030.135} C_VEL
LIN {X 0,Y 559.166,Z 238.453,A -85,B 0,C 180,E1 -3033.172,E2 -3033.172} C_VEL
LIN {X 0,Y 559.151,Z 238.457,A -85,B 0,C 180,E1 -3035.495,E2 -3035.495} C_VEL
LIN {X 0,Y 559.165,Z 238.453,A -85,B 0,C 180,E1 -3038.624,E2 -3038.624} C_VEL
LIN {X 0,Y 559.164,Z 238.453,A -85,B 0,C 180,E1 -3040.926,E2 -3040.926} C_VEL
LIN {X 0,Y 559.165,Z 238.46,A -85,B 0,C 180,E1 -3043.948,E2 -3043.948} C_VEL
LIN {X 0,Y 559.168,Z 238.455,A -85,B 0,C 180,E1 -3046.184,E2 -3046.184} C_VEL
LIN {X 0,Y 559.188,Z 238.45,A -85,B 0,C 180,E1 -3049.134,E2 -3049.134} C_VEL
LIN {X 0,Y 559.2,Z 238.45,A -85,B 0,C 180,E1 -3052.054,E2 -3052.054} C_VEL
LIN {X 0,Y 559.25,Z 238.443,A -85,B 0,C 180,E1 -3054.954,E2 -3054.954} C_VEL
LIN {X 0,Y 559.245,Z 238.448,A -85,B 0,C 180,E1 -3057.84,E2 -3057.84} C_VEL
LIN {X 0,Y 559.268,Z 238.44,A -85,B 0,C 180,E1 -3060.72,E2 -3060.72} C_VEL
LIN {X 0,Y 559.237,Z 238.443,A -85,B 0,C 180,E1 -3062.882,E2 -3062.882} C_VEL
LIN {X 0,Y 559.223,Z 238.449,A -85,B 0,C 180,E1 -3065.771,E2 -3065.771} C_VEL
LIN {X 0,Y 559.186,Z 238.45,A -85,B 0,C 180,E1 -3068.675,E2 -3068.675} C_VEL
LIN {X 0,Y 559.199,Z 238.453,A -85,B 0,C 180,E1 -3071.601,E2 -3071.601} C_VEL
LIN {X 0,Y 559.193,Z 238.45,A -85,B 0,C 180,E1 -3074.596,E2 -3074.596} C_VEL
LIN {X 0,Y 559.158,Z 238.459,A -85,B 0,C 180,E1 -3077.557,E2 -3077.557} C_VEL
LIN {X 0,Y 559.167,Z 238.453,A -85,B 0,C 180,E1 -3079.838,E2 -3079.838} C_VEL
LIN {X 0,Y 559.137,Z 238.456,A -85,B 0,C 180,E1 -3082.153,E2 -3082.153} C_VEL
LIN {X 0,Y 559.174,Z 238.461,A -85,B 0,C 180,E1 -3085.188,E2 -3085.188} C_VEL
LIN {X 0,Y 559.185,Z 238.449,A -85,B 0,C 180,E1 -3087.712,E2 -3087.712} C_VEL
LIN {X 0,Y 559.142,Z 238.457,A -85,B 0,C 180,E1 -3090.623,E2 -3090.623} C_VEL
LIN {X 0,Y 558.483,Z 238.545,A -85,B 0,C 180,E1 -3091.225,E2 -3091.225} C_VEL
LIN {X 0,Y 555.621,Z 238.901,A -85,B 0,C 180,E1 -3092.201,E2 -3092.201} C_VEL
LIN {X 0,Y 553.208,Z 239.204,A -85,B 0,C 180,E1 -3092.987,E2 -3092.987} C_VEL
LIN {X 0,Y 552.187,Z 239.323,A -85,B 0,C 180,E1 -3093.593,E2 -3093.593} C_VEL
LIN {X 0,Y 552.112,Z 239.33,A -85,B 0,C 180,E1 -3093.799,E2 -3093.799} C_VEL
LIN {X 0,Y 552.11,Z 239.336,A -85,B 0,C 180,E1 -3096.747,E2 -3096.747} C_VEL
LIN {X 0,Y 552.131,Z 239.327,A -85,B 0,C 180,E1 -3099.528,E2 -3099.528} C_VEL
LIN {X 0,Y 552.128,Z 239.333,A -85,B 0,C 180,E1 -3102.426,E2 -3102.426} C_VEL
LIN {X 0,Y 552.099,Z 239.334,A -85,B 0,C 180,E1 -3105.564,E2 -3105.564} C_VEL
LIN {X 0,Y 552.138,Z 239.335,A -85,B 0,C 180,E1 -3108.677,E2 -3108.677} C_VEL
LIN {X 0,Y 552.118,Z 239.324,A -85,B 0,C 180,E1 -3111.412,E2 -3111.412} C_VEL
LIN {X 0,Y 552.086,Z 239.338,A -85,B 0,C 180,E1 -3114.157,E2 -3114.157} C_VEL
LIN {X 0,Y 552.109,Z 239.338,A -85,B 0,C 180,E1 -3116.814,E2 -3116.814} C_VEL
LIN {X 0,Y 552.102,Z 239.334,A -85,B 0,C 180,E1 -3119.391,E2 -3119.391} C_VEL
LIN {X 0,Y 552.109,Z 239.333,A -85,B 0,C 180,E1 -3121.902,E2 -3121.902} C_VEL
LIN {X 0,Y 552.179,Z 239.471,A -85,B 0,C 180,E1 -3122.928,E2 -3122.928} C_VEL
LIN {X 0,Y 553.571,Z 246.479,A -85,B 0,C 180,E1 -3124.024,E2 -3124.024} C_VEL
LIN {X 0,Y 553.248,Z 264.912,A -85,B 0,C 180,E1 -3126.638,E2 -3126.638} C_VEL
LIN {X 0,Y 552.893,Z 284.297,A -85,B 0,C 180,E1 -3129.345,E2 -3129.345} C_VEL
LIN {X 0,Y 552.559,Z 306.873,A -85,B 0,C 180,E1 -3132.451,E2 -3132.451} C_VEL
LIN {X 0,Y 552.443,Z 315.243,A -85,B 0,C 180,E1 -3133.581,E2 -3133.581} C_VEL
LIN {X 0,Y 553.338,Z 321.795,A -85,B 0,C 180,E1 -3133.767,E2 -3133.767} C_VEL
LIN {X 0,Y 553.156,Z 424.658,A -85,B 0,C 180,E1 -3135.133,E2 -3135.133} C_VEL
LIN {X 0,Y 553.025,Z 437.358,A -85,B 0,C 180,E1 -3135.441,E2 -3135.441} C_VEL
LIN {X 0,Y 552.888,Z 449.673,A -85,B 0,C 180,E1 -3135.883,E2 -3135.883} C_VEL
LIN {X 0,Y 552.663,Z 462.053,A -85,B 0,C 180,E1 -3136.487,E2 -3136.487} C_VEL
LIN {X 0,Y 552.444,Z 473.703,A -85,B 0,C 180,E1 -3137.23,E2 -3137.23} C_VEL
LIN {X 0,Y 552.263,Z 484.169,A -85,B 0,C 180,E1 -3138.066,E2 -3138.066} C_VEL
LIN {X 0,Y 552.082,Z 493.567,A -85,B 0,C 180,E1 -3138.992,E2 -3138.992} C_VEL
LIN {X 0,Y 551.968,Z 502.633,A -85,B 0,C 180,E1 -3140.102,E2 -3140.102} C_VEL
LIN {X 0,Y 551.857,Z 509.927,A -85,B 0,C 180,E1 -3141.21,E2 -3141.21} C_VEL
LIN {X 0,Y 551.81,Z 515.759,A -85,B 0,C 180,E1 -3142.315,E2 -3142.315} C_VEL
LIN {X 0,Y 551.767,Z 520.53,A -85,B 0,C 180,E1 -3143.471,E2 -3143.471} C_VEL
LIN {X 0,Y 551.758,Z 522.756,A -85,B 0,C 180,E1 -3144.151,E2 -3144.151} C_VEL
LIN {X 0,Y 551.695,Z 524.733,A -85,B 0,C 180,E1 -3144.884,E2 -3144.884} C_VEL
LIN {X 0,Y 551.703,Z 526.294,A -85,B 0,C 180,E1 -3145.617,E2 -3145.617} C_VEL
LIN {X 0,Y 551.733,Z 527.426,A -85,B 0,C 180,E1 -3146.348,E2 -3146.348} C_VEL
LIN {X 0,Y 551.719,Z 528.132,A -85,B 0,C 180,E1 -3147.079,E2 -3147.079} C_VEL
LIN {X 0,Y 551.644,Z 528.399,A -85,B 0,C 180,E1 -3148.54,E2 -3148.54} C_VEL
LIN {X 0,Y 551.641,Z 527.94,A -85,B 0,C 180,E1 -3149.27,E2 -3149.27} C_VEL
LIN {X 0,Y 551.645,Z 525.786,A -85,B 0,C 180,E1 -3150.73,E2 -3150.73} C_VEL
LIN {X 0,Y 551.742,Z 523.087,A -85,B 0,C 180,E1 -3151.825,E2 -3151.825} C_VEL
LIN {X 0,Y 551.752,Z 519.381,A -85,B 0,C 180,E1 -3152.92,E2 -3152.92} C_VEL
LIN {X 0,Y 551.822,Z 514.57,A -85,B 0,C 180,E1 -3154.017,E2 -3154.017} C_VEL
LIN {X 0,Y 551.899,Z 508.504,A -85,B 0,C 180,E1 -3155.114,E2 -3155.114} C_VEL
LIN {X 0,Y 552.033,Z 500.971,A -85,B 0,C 180,E1 -3156.212,E2 -3156.212} C_VEL
LIN {X 0,Y 552.123,Z 492.726,A -85,B 0,C 180,E1 -3157.189,E2 -3157.189} C_VEL
LIN {X 0,Y 552.311,Z 482.847,A -85,B 0,C 180,E1 -3158.138,E2 -3158.138} C_VEL
LIN {X 0,Y 552.512,Z 472.228,A -85,B 0,C 180,E1 -3158.964,E2 -3158.964} C_VEL
LIN {X 0,Y 552.702,Z 461.96,A -85,B 0,C 180,E1 -3159.607,E2 -3159.607} C_VEL
LIN {X 0,Y 552.859,Z 450.849,A -85,B 0,C 180,E1 -3160.159,E2 -3160.159} C_VEL
LIN {X 0,Y 553.006,Z 437.616,A -85,B 0,C 180,E1 -3160.642,E2 -3160.642} C_VEL
LIN {X 0,Y 553.119,Z 424.378,A -85,B 0,C 180,E1 -3160.964,E2 -3160.964} C_VEL
LIN {X 0,Y 553.317,Z 321.481,A -85,B 0,C 180,E1 -3162.328,E2 -3162.328} C_VEL
LIN {X 0,Y 552.465,Z 315.601,A -85,B 0,C 180,E1 -3162.489,E2 -3162.489} C_VEL
LIN {X 0,Y 552.505,Z 312.555,A -85,B 0,C 180,E1 -3162.862,E2 -3162.862} C_VEL
LIN {X 0,Y 552.792,Z 290.696,A -85,B 0,C 180,E1 -3165.863,E2 -3165.863} C_VEL
LIN {X 0,Y 553.145,Z 270.194,A -85,B 0,C 180,E1 -3168.712,E2 -3168.712} C_VEL
LIN {X 0,Y 553.605,Z 248.602,A -85,B 0,C 180,E1 -3171.76,E2 -3171.76} C_VEL
LIN {X 0,Y 553.172,Z 244.257,A -85,B 0,C 180,E1 -3172.404,E2 -3172.404} C_VEL
LIN {X 0,Y 552.124,Z 239.407,A -85,B 0,C 180,E1 -3173.191,E2 -3173.191} C_VEL
LIN {X 0,Y 552.133,Z 239.317,A -85,B 0,C 180,E1 -3175.644,E2 -3175.644} C_VEL
LIN {X 0,Y 552.127,Z 239.331,A -85,B 0,C 180,E1 -3178.561,E2 -3178.561} C_VEL
LIN {X 0,Y 552.113,Z 239.341,A -85,B 0,C 180,E1 -3181.475,E2 -3181.475} C_VEL
LIN {X 0,Y 552.134,Z 239.326,A -85,B 0,C 180,E1 -3184.169,E2 -3184.169} C_VEL
LIN {X 0,Y 552.106,Z 239.335,A -85,B 0,C 180,E1 -3186.746,E2 -3186.746} C_VEL
LIN {X 0,Y 552.128,Z 239.335,A -85,B 0,C 180,E1 -3189.526,E2 -3189.526} C_VEL
LIN {X 0,Y 552.131,Z 239.329,A -85,B 0,C 180,E1 -3192.424,E2 -3192.424} C_VEL
LIN {X 0,Y 552.096,Z 239.336,A -85,B 0,C 180,E1 -3195.562,E2 -3195.562} C_VEL
LIN {X 0,Y 552.13,Z 239.332,A -85,B 0,C 180,E1 -3198.676,E2 -3198.676} C_VEL
LIN {X 0,Y 552.118,Z 239.335,A -85,B 0,C 180,E1 -3201.41,E2 -3201.41} C_VEL
LIN {X 0,Y 552.11,Z 239.331,A -85,B 0,C 180,E1 -3204.158,E2 -3204.158} C_VEL
LIN {X 0,Y 552.119,Z 239.331,A -85,B 0,C 180,E1 -3206.814,E2 -3206.814} C_VEL
LIN {X 0,Y 552.11,Z 239.335,A -85,B 0,C 180,E1 -3209.391,E2 -3209.391} C_VEL
LIN {X 0,Y 552.118,Z 239.329,A -85,B 0,C 180,E1 -3211.902,E2 -3211.902} C_VEL
LIN {X 0,Y 552.15,Z 239.333,A -85,B 0,C 180,E1 -3214.649,E2 -3214.649} C_VEL
LIN {X 0,Y 552.09,Z 239.335,A -85,B 0,C 180,E1 -3217.549,E2 -3217.549} C_VEL
LIN {X 0,Y 552.151,Z 239.333,A -85,B 0,C 180,E1 -3220.674,E2 -3220.674} C_VEL
LIN {X 0,Y 552.114,Z 239.331,A -85,B 0,C 180,E1 -3223.737,E2 -3223.737} C_VEL
LIN {X 0,Y 552.131,Z 239.328,A -85,B 0,C 180,E1 -3226.004,E2 -3226.004} C_VEL
LIN {X 0,Y 552.155,Z 239.329,A -85,B 0,C 180,E1 -3228.993,E2 -3228.993} C_VEL
LIN {X 0,Y 552.154,Z 239.327,A -85,B 0,C 180,E1 -3231.951,E2 -3231.951} C_VEL
LIN {X 0,Y 552.224,Z 239.319,A -85,B 0,C 180,E1 -3234.889,E2 -3234.889} C_VEL
LIN {X 0,Y 552.216,Z 239.319,A -85,B 0,C 180,E1 -3237.812,E2 -3237.812} C_VEL
LIN {X 0,Y 552.239,Z 239.319,A -85,B 0,C 180,E1 -3240.729,E2 -3240.729} C_VEL
LIN {X 0,Y 552.202,Z 239.323,A -85,B 0,C 180,E1 -3242.918,E2 -3242.918} C_VEL
LIN {X 0,Y 552.194,Z 239.322,A -85,B 0,C 180,E1 -3245.844,E2 -3245.844} C_VEL
LIN {X 0,Y 552.156,Z 239.328,A -85,B 0,C 180,E1 -3248.786,E2 -3248.786} C_VEL
LIN {X 0,Y 552.155,Z 239.326,A -85,B 0,C 180,E1 -3251.75,E2 -3251.75} C_VEL
LIN {X 0,Y 552.129,Z 239.33,A -85,B 0,C 180,E1 -3254.748,E2 -3254.748} C_VEL
LIN {X 0,Y 552.108,Z 239.335,A -85,B 0,C 180,E1 -3257.788,E2 -3257.788} C_VEL
LIN {X 0,Y 552.124,Z 239.338,A -85,B 0,C 180,E1 -3260.101,E2 -3260.101} C_VEL
LIN {X 0,Y 552.089,Z 239.339,A -85,B 0,C 180,E1 -3262.451,E2 -3262.451} C_VEL
LIN {X 0,Y 552.148,Z 239.326,A -85,B 0,C 180,E1 -3265.351,E2 -3265.351} C_VEL
LIN {X 0,Y 552.119,Z 239.336,A -85,B 0,C 180,E1 -3268.098,E2 -3268.098} C_VEL
LIN {X 0,Y 552.108,Z 239.329,A -85,B 0,C 180,E1 -3270.609,E2 -3270.609} C_VEL
LIN {X 0,Y 552.117,Z 239.331,A -85,B 0,C 180,E1 -3273.186,E2 -3273.186} C_VEL
LIN {X 0,Y 552.108,Z 239.338,A -85,B 0,C 180,E1 -3275.842,E2 -3275.842} C_VEL
LIN {X 0,Y 552.121,Z 239.331,A -85,B 0,C 180,E1 -3279.062,E2 -3279.062} C_VEL
LIN {X 0,Y 552.135,Z 239.333,A -85,B 0,C 180,E1 -3281.445,E2 -3281.445} C_VEL
LIN {X 0,Y 552.091,Z 239.335,A -85,B 0,C 180,E1 -3284.532,E2 -3284.532} C_VEL
LIN {X 0,Y 552.127,Z 239.329,A -85,B 0,C 180,E1 -3287.585,E2 -3287.585} C_VEL
LIN {X 0,Y 552.126,Z 239.33,A -85,B 0,C 180,E1 -3290.473,E2 -3290.473} C_VEL
LIN {X 0,Y 552.103,Z 239.337,A -85,B 0,C 180,E1 -3293.318,E2 -3293.318} C_VEL
LIN {X 0,Y 552.125,Z 239.335,A -85,B 0,C 180,E1 -3295.94,E2 -3295.94} C_VEL
LIN {X 0,Y 552.117,Z 239.327,A -85,B 0,C 180,E1 -3298.541,E2 -3298.541} C_VEL
LIN {X 0,Y 552.123,Z 239.334,A -85,B 0,C 180,E1 -3301.438,E2 -3301.438} C_VEL
LIN {X 0,Y 552.13,Z 239.332,A -85,B 0,C 180,E1 -3304.356,E2 -3304.356} C_VEL
LIN {X 0,Y 552.18,Z 239.55,A -85,B 0,C 180,E1 -3305.741,E2 -3305.741} C_VEL
LIN {X 0,Y 553.888,Z 247.564,A -85,B 0,C 180,E1 -3306.838,E2 -3306.838} C_VEL
LIN {X 0,Y 553.369,Z 271.297,A -85,B 0,C 180,E1 -3309.752,E2 -3309.752} C_VEL
LIN {X 0,Y 552.874,Z 294.58,A -85,B 0,C 180,E1 -3312.549,E2 -3312.549} C_VEL
LIN {X 0,Y 553.206,Z 296.868,A -85,B 0,C 180,E1 -3312.629,E2 -3312.629} C_VEL
LIN {X 0,Y 554.209,Z 303.023,A -85,B 0,C 180,E1 -3312.74,E2 -3312.74} C_VEL
LIN {X 0,Y 553.778,Z 432.652,A -85,B 0,C 180,E1 -3314.449,E2 -3314.449} C_VEL
LIN {X 0,Y 553.611,Z 446.81,A -85,B 0,C 180,E1 -3314.773,E2 -3314.773} C_VEL
LIN {X 0,Y 553.43,Z 460.577,A -85,B 0,C 180,E1 -3315.24,E2 -3315.24} C_VEL
LIN {X 0,Y 553.2,Z 473.878,A -85,B 0,C 180,E1 -3315.845,E2 -3315.845} C_VEL
LIN {X 0,Y 552.871,Z 486.677,A -85,B 0,C 180,E1 -3316.586,E2 -3316.586} C_VEL
LIN {X 0,Y 552.645,Z 498.31,A -85,B 0,C 180,E1 -3317.422,E2 -3317.422} C_VEL
LIN {X 0,Y 552.413,Z 509.651,A -85,B 0,C 180,E1 -3318.414,E2 -3318.414} C_VEL
LIN {X 0,Y 552.227,Z 520.335,A -85,B 0,C 180,E1 -3319.552,E2 -3319.552} C_VEL
LIN {X 0,Y 552.073,Z 528.912,A -85,B 0,C 180,E1 -3320.659,E2 -3320.659} C_VEL
LIN {X 0,Y 551.901,Z 537.119,A -85,B 0,C 180,E1 -3321.948,E2 -3321.948} C_VEL
LIN {X 0,Y 551.823,Z 542.864,A -85,B 0,C 180,E1 -3323.051,E2 -3323.051} C_VEL
LIN {X 0,Y 551.792,Z 548.961,A -85,B 0,C 180,E1 -3324.519,E2 -3324.519} C_VEL
LIN {X 0,Y 551.759,Z 552.444,A -85,B 0,C 180,E1 -3325.617,E2 -3325.617} C_VEL
LIN {X 0,Y 551.72,Z 555.832,A -85,B 0,C 180,E1 -3327.079,E2 -3327.079} C_VEL
LIN {X 0,Y 551.64,Z 557.834,A -85,B 0,C 180,E1 -3328.54,E2 -3328.54} C_VEL
LIN {X 0,Y 551.639,Z 558.5,A -85,B 0,C 180,E1 -3330,E2 -3330} C_VEL
LIN {X 0,Y 551.64,Z 557.835,A -85,B 0,C 180,E1 -3331.46,E2 -3331.46} C_VEL
LIN {X 0,Y 551.72,Z 555.835,A -85,B 0,C 180,E1 -3332.921,E2 -3332.921} C_VEL
LIN {X 0,Y 551.759,Z 552.447,A -85,B 0,C 180,E1 -3334.383,E2 -3334.383} C_VEL
LIN {X 0,Y 551.823,Z 547.568,A -85,B 0,C 180,E1 -3335.848,E2 -3335.848} C_VEL
LIN {X 0,Y 551.832,Z 541.055,A -85,B 0,C 180,E1 -3337.317,E2 -3337.317} C_VEL
LIN {X 0,Y 551.962,Z 533.804,A -85,B 0,C 180,E1 -3338.604,E2 -3338.604} C_VEL
LIN {X 0,Y 552.116,Z 524.823,A -85,B 0,C 180,E1 -3339.895,E2 -3339.895} C_VEL
LIN {X 0,Y 552.346,Z 515.394,A -85,B 0,C 180,E1 -3341.003,E2 -3341.003} C_VEL
LIN {X 0,Y 552.538,Z 504.954,A -85,B 0,C 180,E1 -3342.021,E2 -3342.021} C_VEL
LIN {X 0,Y 552.76,Z 493.431,A -85,B 0,C 180,E1 -3342.949,E2 -3342.949} C_VEL
LIN {X 0,Y 553.012,Z 480.642,A -85,B 0,C 180,E1 -3343.785,E2 -3343.785} C_VEL
LIN {X 0,Y 553.283,Z 468.149,A -85,B 0,C 180,E1 -3344.435,E2 -3344.435} C_VEL
LIN {X 0,Y 553.533,Z 454.108,A -85,B 0,C 180,E1 -3344.997,E2 -3344.997} C_VEL
LIN {X 0,Y 553.689,Z 439.869,A -85,B 0,C 180,E1 -3345.405,E2 -3345.405} C_VEL
LIN {X 0,Y 553.799,Z 424.842,A -85,B 0,C 180,E1 -3345.668,E2 -3345.668} C_VEL
LIN {X 0,Y 554.142,Z 302.143,A -85,B 0,C 180,E1 -3347.273,E2 -3347.273} C_VEL
LIN {X 0,Y 552.915,Z 294.951,A -85,B 0,C 180,E1 -3347.426,E2 -3347.426} C_VEL
LIN {X 0,Y 553.255,Z 274.893,A -85,B 0,C 180,E1 -3349.811,E2 -3349.811} C_VEL
LIN {X 0,Y 553.817,Z 250.743,A -85,B 0,C 180,E1 -3352.771,E2 -3352.771} C_VEL
LIN {X 0,Y 553.769,Z 246.426,A -85,B 0,C 180,E1 -3353.31,E2 -3353.31} C_VEL
LIN {X 0,Y 552.138,Z 239.401,A -85,B 0,C 180,E1 -3354.311,E2 -3354.311} C_VEL
LIN {X 0,Y 552.139,Z 239.332,A -85,B 0,C 180,E1 -3357.273,E2 -3357.273} C_VEL
LIN {X 0,Y 552.116,Z 239.335,A -85,B 0,C 180,E1 -3360.05,E2 -3360.05} C_VEL
LIN {X 0,Y 552.127,Z 239.334,A -85,B 0,C 180,E1 -3362.848,E2 -3362.848} C_VEL
LIN {X 0,Y 552.075,Z 239.334,A -85,B 0,C 180,E1 -3365.439,E2 -3365.439} C_VEL
LIN {X 0,Y 552.094,Z 239.333,A -85,B 0,C 180,E1 -3367.885,E2 -3367.885} C_VEL
LIN {X 0,Y 552.107,Z 239.338,A -85,B 0,C 180,E1 -3370.48,E2 -3370.48} C_VEL
LIN {X 0,Y 552.111,Z 239.332,A -85,B 0,C 180,E1 -3373.484,E2 -3373.484} C_VEL
LIN {X 0,Y 552.103,Z 239.337,A -85,B 0,C 180,E1 -3376.576,E2 -3376.576} C_VEL
LIN {X 0,Y 552.118,Z 239.329,A -85,B 0,C 180,E1 -3379.52,E2 -3379.52} C_VEL
LIN {X 0,Y 552.089,Z 239.339,A -85,B 0,C 180,E1 -3382.336,E2 -3382.336} C_VEL
LIN {X 0,Y 552.124,Z 239.328,A -85,B 0,C 180,E1 -3385.054,E2 -3385.054} C_VEL
LIN {X 0,Y 552.122,Z 239.334,A -85,B 0,C 180,E1 -3387.682,E2 -3387.682} C_VEL
LIN {X 0,Y 552.139,Z 239.33,A -85,B 0,C 180,E1 -3390.237,E2 -3390.237} C_VEL
LIN {X 0,Y 552.135,Z 239.328,A -85,B 0,C 180,E1 -3392.999,E2 -3392.999} C_VEL
LIN {X 0,Y 552.107,Z 239.332,A -85,B 0,C 180,E1 -3395.161,E2 -3395.161} C_VEL
LIN {X 0,Y 552.09,Z 239.338,A -85,B 0,C 180,E1 -3397.549,E2 -3397.549} C_VEL
LIN {X 0,Y 552.15,Z 239.327,A -85,B 0,C 180,E1 -3400.674,E2 -3400.674} C_VEL
LIN {X 0,Y 552.114,Z 239.338,A -85,B 0,C 180,E1 -3403.737,E2 -3403.737} C_VEL
LIN {X 0,Y 552.131,Z 239.335,A -85,B 0,C 180,E1 -3406.005,E2 -3406.005} C_VEL
LIN {X 0,Y 552.155,Z 239.325,A -85,B 0,C 180,E1 -3408.993,E2 -3408.993} C_VEL
LIN {X 0,Y 552.154,Z 239.329,A -85,B 0,C 180,E1 -3411.952,E2 -3411.952} C_VEL
LIN {X 0,Y 552.224,Z 239.318,A -85,B 0,C 180,E1 -3414.889,E2 -3414.889} C_VEL
LIN {X 0,Y 552.216,Z 239.323,A -85,B 0,C 180,E1 -3417.812,E2 -3417.812} C_VEL
LIN {X 0,Y 552.238,Z 239.316,A -85,B 0,C 180,E1 -3420.729,E2 -3420.729} C_VEL
LIN {X 0,Y 552.203,Z 239.32,A -85,B 0,C 180,E1 -3422.918,E2 -3422.918} C_VEL
LIN {X 0,Y 552.194,Z 239.323,A -85,B 0,C 180,E1 -3425.844,E2 -3425.844} C_VEL
LIN {X 0,Y 552.157,Z 239.327,A -85,B 0,C 180,E1 -3428.786,E2 -3428.786} C_VEL
LIN {X 0,Y 552.156,Z 239.328,A -85,B 0,C 180,E1 -3431.751,E2 -3431.751} C_VEL
LIN {X 0,Y 552.13,Z 239.331,A -85,B 0,C 180,E1 -3434.749,E2 -3434.749} C_VEL
LIN {X 0,Y 552.109,Z 239.334,A -85,B 0,C 180,E1 -3437.789,E2 -3437.789} C_VEL
LIN {X 0,Y 552.126,Z 239.328,A -85,B 0,C 180,E1 -3440.102,E2 -3440.102} C_VEL
LIN {X 0,Y 552.091,Z 239.335,A -85,B 0,C 180,E1 -3442.451,E2 -3442.451} C_VEL
LIN {X 0,Y 552.151,Z 239.333,A -85,B 0,C 180,E1 -3445.351,E2 -3445.351} C_VEL
LIN {X 0,Y 552.119,Z 239.327,A -85,B 0,C 180,E1 -3448.098,E2 -3448.098} C_VEL
LIN {X 0,Y 552.103,Z 239.333,A -85,B 0,C 180,E1 -3450.619,E2 -3450.619} C_VEL
LIN {X 0,Y 552.12,Z 239.335,A -85,B 0,C 180,E1 -3453.186,E2 -3453.186} C_VEL
LIN {X 0,Y 552.112,Z 239.33,A -85,B 0,C 180,E1 -3453.799,E2 -3453.799} C_VEL
LIN {X 0,Y 551.477,Z 239.411,A -85,B 0,C 180,E1 -3454.407,E2 -3454.407} C_VEL
LIN {X 0,Y 548.655,Z 239.768,A -85,B 0,C 180,E1 -3455.396,E2 -3455.396} C_VEL
LIN {X 0,Y 546.234,Z 240.074,A -85,B 0,C 180,E1 -3456.191,E2 -3456.191} C_VEL
LIN {X 0,Y 545.165,Z 240.205,A -85,B 0,C 180,E1 -3456.805,E2 -3456.805} C_VEL
LIN {X 0,Y 545.063,Z 240.216,A -85,B 0,C 180,E1 -3457.013,E2 -3457.013} C_VEL
LIN {X 0,Y 545.07,Z 240.205,A -85,B 0,C 180,E1 -3460.143,E2 -3460.143} C_VEL
LIN {X 0,Y 545.077,Z 240.211,A -85,B 0,C 180,E1 -3463.107,E2 -3463.107} C_VEL
LIN {X 0,Y 545.065,Z 240.212,A -85,B 0,C 180,E1 -3466.225,E2 -3466.225} C_VEL
LIN {X 0,Y 545.094,Z 240.214,A -85,B 0,C 180,E1 -3468.887,E2 -3468.887} C_VEL
LIN {X 0,Y 545.052,Z 240.203,A -85,B 0,C 180,E1 -3471.763,E2 -3471.763} C_VEL
LIN {X 0,Y 545.037,Z 240.222,A -85,B 0,C 180,E1 -3474.532,E2 -3474.532} C_VEL
LIN {X 0,Y 545.067,Z 240.213,A -85,B 0,C 180,E1 -3477.212,E2 -3477.212} C_VEL
LIN {X 0,Y 545.063,Z 240.211,A -85,B 0,C 180,E1 -3479.811,E2 -3479.811} C_VEL
LIN {X 0,Y 545.157,Z 240.391,A -85,B 0,C 180,E1 -3482.73,E2 -3482.73} C_VEL
LIN {X 0,Y 546.768,Z 249.331,A -85,B 0,C 180,E1 -3484.128,E2 -3484.128} C_VEL
LIN {X 0,Y 546.313,Z 268.705,A -85,B 0,C 180,E1 -3486.899,E2 -3486.899} C_VEL
LIN {X 0,Y 545.821,Z 290.091,A -85,B 0,C 180,E1 -3489.911,E2 -3489.911} C_VEL
LIN {X 0,Y 545.507,Z 310.617,A -85,B 0,C 180,E1 -3492.764,E2 -3492.764} C_VEL
LIN {X 0,Y 545.497,Z 315.501,A -85,B 0,C 180,E1 -3493.414,E2 -3493.414} C_VEL
LIN {X 0,Y 546.065,Z 319.563,A -85,B 0,C 180,E1 -3493.522,E2 -3493.522} C_VEL
LIN {X 0,Y 546.612,Z 325.517,A -85,B 0,C 180,E1 -3493.617,E2 -3493.617} C_VEL
LIN {X 0,Y 546.293,Z 425.213,A -85,B 0,C 180,E1 -3494.955,E2 -3494.955} C_VEL
LIN {X 0,Y 546.151,Z 438.011,A -85,B 0,C 180,E1 -3495.277,E2 -3495.277} C_VEL
LIN {X 0,Y 545.974,Z 450.667,A -85,B 0,C 180,E1 -3495.748,E2 -3495.748} C_VEL
LIN {X 0,Y 545.741,Z 461.911,A -85,B 0,C 180,E1 -3496.312,E2 -3496.312} C_VEL
LIN {X 0,Y 545.479,Z 473.521,A -85,B 0,C 180,E1 -3497.064,E2 -3497.064} C_VEL
LIN {X 0,Y 545.246,Z 483.952,A -85,B 0,C 180,E1 -3497.91,E2 -3497.91} C_VEL
LIN {X 0,Y 545.045,Z 493.342,A -85,B 0,C 180,E1 -3498.848,E2 -3498.848} C_VEL
LIN {X 0,Y 544.939,Z 502.445,A -85,B 0,C 180,E1 -3499.973,E2 -3499.973} C_VEL
LIN {X 0,Y 544.804,Z 509.772,A -85,B 0,C 180,E1 -3501.095,E2 -3501.095} C_VEL
LIN {X 0,Y 544.744,Z 515.637,A -85,B 0,C 180,E1 -3502.215,E2 -3502.215} C_VEL
LIN {X 0,Y 544.669,Z 520.806,A -85,B 0,C 180,E1 -3503.494,E2 -3503.494} C_VEL
LIN {X 0,Y 544.616,Z 524.671,A -85,B 0,C 180,E1 -3504.817,E2 -3504.817} C_VEL
LIN {X 0,Y 544.6,Z 526.245,A -85,B 0,C 180,E1 -3505.559,E2 -3505.559} C_VEL
LIN {X 0,Y 544.647,Z 527.397,A -85,B 0,C 180,E1 -3506.301,E2 -3506.301} C_VEL
LIN {X 0,Y 544.646,Z 528.115,A -85,B 0,C 180,E1 -3507.041,E2 -3507.041} C_VEL
LIN {X 0,Y 544.545,Z 528.404,A -85,B 0,C 180,E1 -3508.521,E2 -3508.521} C_VEL
LIN {X 0,Y 544.542,Z 527.966,A -85,B 0,C 180,E1 -3509.26,E2 -3509.26} C_VEL
LIN {X 0,Y 544.544,Z 527.098,A -85,B 0,C 180,E1 -3510,E2 -3510} C_VEL
LIN {X 0,Y 544.572,Z 524.173,A -85,B 0,C 180,E1 -3511.479,E2 -3511.479} C_VEL
LIN {X 0,Y 544.658,Z 520.829,A -85,B 0,C 180,E1 -3512.588,E2 -3512.588} C_VEL
LIN {X 0,Y 544.727,Z 516.427,A -85,B 0,C 180,E1 -3513.699,E2 -3513.699} C_VEL
LIN {X 0,Y 544.864,Z 509.771,A -85,B 0,C 180,E1 -3514.995,E2 -3514.995} C_VEL
LIN {X 0,Y 544.94,Z 502.523,A -85,B 0,C 180,E1 -3516.106,E2 -3516.106} C_VEL
LIN {X 0,Y 545.076,Z 493.509,A -85,B 0,C 180,E1 -3517.222,E2 -3517.222} C_VEL
LIN {X 0,Y 545.287,Z 484.282,A -85,B 0,C 180,E1 -3518.15,E2 -3518.15} C_VEL
LIN {X 0,Y 545.499,Z 474.04,A -85,B 0,C 180,E1 -3518.987,E2 -3518.987} C_VEL
LIN {X 0,Y 545.743,Z 462.681,A -85,B 0,C 180,E1 -3519.731,E2 -3519.731} C_VEL
LIN {X 0,Y 545.945,Z 450.827,A -85,B 0,C 180,E1 -3520.336,E2 -3520.336} C_VEL
LIN {X 0,Y 546.105,Z 437.664,A -85,B 0,C 180,E1 -3520.825,E2 -3520.825} C_VEL
LIN {X 0,Y 546.265,Z 424.497,A -85,B 0,C 180,E1 -3521.15,E2 -3521.15} C_VEL
LIN {X 0,Y 546.496,Z 322.291,A -85,B 0,C 180,E1 -3522.518,E2 -3522.518} C_VEL
LIN {X 0,Y 545.498,Z 315.876,A -85,B 0,C 180,E1 -3522.651,E2 -3522.651} C_VEL
LIN {X 0,Y 545.509,Z 312.751,A -85,B 0,C 180,E1 -3523.03,E2 -3523.03} C_VEL
LIN {X 0,Y 545.83,Z 292.243,A -85,B 0,C 180,E1 -3525.879,E2 -3525.879} C_VEL
LIN {X 0,Y 546.217,Z 271.734,A -85,B 0,C 180,E1 -3528.763,E2 -3528.763} C_VEL
LIN {X 0,Y 546.745,Z 249.865,A -85,B 0,C 180,E1 -3531.886,E2 -3531.886} C_VEL
LIN {X 0,Y 545.979,Z 244.423,A -85,B 0,C 180,E1 -3532.716,E2 -3532.716} C_VEL
LIN {X 0,Y 545.095,Z 240.28,A -85,B 0,C 180,E1 -3533.407,E2 -3533.407} C_VEL
LIN {X 0,Y 545.082,Z 240.198,A -85,B 0,C 180,E1 -3536,E2 -3536} C_VEL
LIN {X 0,Y 545.092,Z 240.209,A -85,B 0,C 180,E1 -3538.747,E2 -3538.747} C_VEL
LIN {X 0,Y 545.061,Z 240.215,A -85,B 0,C 180,E1 -3541.678,E2 -3541.678} C_VEL
LIN {X 0,Y 545.076,Z 240.204,A -85,B 0,C 180,E1 -3544.391,E2 -3544.391} C_VEL
LIN {X 0,Y 545.036,Z 240.22,A -85,B 0,C 180,E1 -3547.303,E2 -3547.303} C_VEL
LIN {X 0,Y 545.066,Z 240.209,A -85,B 0,C 180,E1 -3550.142,E2 -3550.142} C_VEL
LIN {X 0,Y 545.086,Z 240.214,A -85,B 0,C 180,E1 -3553.105,E2 -3553.105} C_VEL
LIN {X 0,Y 545.049,Z 240.21,A -85,B 0,C 180,E1 -3556.225,E2 -3556.225} C_VEL
LIN {X 0,Y 545.089,Z 240.212,A -85,B 0,C 180,E1 -3558.885,E2 -3558.885} C_VEL
LIN {X 0,Y 545.052,Z 240.212,A -85,B 0,C 180,E1 -3561.762,E2 -3561.762} C_VEL
LIN {X 0,Y 545.062,Z 240.212,A -85,B 0,C 180,E1 -3564.533,E2 -3564.533} C_VEL
LIN {X 0,Y 545.078,Z 240.212,A -85,B 0,C 180,E1 -3567.212,E2 -3567.212} C_VEL
LIN {X 0,Y 545.098,Z 240.206,A -85,B 0,C 180,E1 -3569.812,E2 -3569.812} C_VEL
LIN {X 0,Y 545.091,Z 240.213,A -85,B 0,C 180,E1 -3572.825,E2 -3572.825} C_VEL
LIN {X 0,Y 545.047,Z 240.21,A -85,B 0,C 180,E1 -3575.63,E2 -3575.63} C_VEL
LIN {X 0,Y 545.061,Z 240.218,A -85,B 0,C 180,E1 -3578.836,E2 -3578.836} C_VEL
LIN {X 0,Y 545.078,Z 240.211,A -85,B 0,C 180,E1 -3581.195,E2 -3581.195} C_VEL
LIN {X 0,Y 545.07,Z 240.209,A -85,B 0,C 180,E1 -3583.521,E2 -3583.521} C_VEL
LIN {X 0,Y 545.089,Z 240.205,A -85,B 0,C 180,E1 -3585.819,E2 -3585.819} C_VEL
LIN {X 0,Y 545.111,Z 240.208,A -85,B 0,C 180,E1 -3588.849,E2 -3588.849} C_VEL
LIN {X 0,Y 545.124,Z 240.202,A -85,B 0,C 180,E1 -3591.847,E2 -3591.847} C_VEL
LIN {X 0,Y 545.2,Z 240.195,A -85,B 0,C 180,E1 -3594.823,E2 -3594.823} C_VEL
LIN {X 0,Y 545.188,Z 240.195,A -85,B 0,C 180,E1 -3597.783,E2 -3597.783} C_VEL
LIN {X 0,Y 545.208,Z 240.195,A -85,B 0,C 180,E1 -3600.738,E2 -3600.738} C_VEL
LIN {X 0,Y 545.168,Z 240.199,A -85,B 0,C 180,E1 -3602.956,E2 -3602.956} C_VEL
LIN {X 0,Y 545.165,Z 240.198,A -85,B 0,C 180,E1 -3605.919,E2 -3605.919} C_VEL
LIN {X 0,Y 545.115,Z 240.204,A -85,B 0,C 180,E1 -3608.9,E2 -3608.9} C_VEL
LIN {X 0,Y 545.127,Z 240.203,A -85,B 0,C 180,E1 -3611.904,E2 -3611.904} C_VEL
LIN {X 0,Y 545.078,Z 240.207,A -85,B 0,C 180,E1 -3614.944,E2 -3614.944} C_VEL
LIN {X 0,Y 545.076,Z 240.215,A -85,B 0,C 180,E1 -3618.026,E2 -3618.026} C_VEL
LIN {X 0,Y 545.088,Z 240.211,A -85,B 0,C 180,E1 -3620.372,E2 -3620.372} C_VEL
LIN {X 0,Y 545.085,Z 240.209,A -85,B 0,C 180,E1 -3623.559,E2 -3623.559} C_VEL
LIN {X 0,Y 545.073,Z 240.216,A -85,B 0,C 180,E1 -3626.001,E2 -3626.001} C_VEL
LIN {X 0,Y 545.085,Z 240.205,A -85,B 0,C 180,E1 -3628.749,E2 -3628.749} C_VEL
LIN {X 0,Y 545.072,Z 240.209,A -85,B 0,C 180,E1 -3631.683,E2 -3631.683} C_VEL
LIN {X 0,Y 545.076,Z 240.209,A -85,B 0,C 180,E1 -3634.563,E2 -3634.563} C_VEL
LIN {X 0,Y 545.034,Z 240.21,A -85,B 0,C 180,E1 -3637.304,E2 -3637.304} C_VEL
LIN {X 0,Y 545.07,Z 240.213,A -85,B 0,C 180,E1 -3640.142,E2 -3640.142} C_VEL
LIN {X 0,Y 545.074,Z 240.207,A -85,B 0,C 180,E1 -3643.107,E2 -3643.107} C_VEL
LIN {X 0,Y 545.063,Z 240.207,A -85,B 0,C 180,E1 -3646.225,E2 -3646.225} C_VEL
LIN {X 0,Y 545.084,Z 240.199,A -85,B 0,C 180,E1 -3648.887,E2 -3648.887} C_VEL
LIN {X 0,Y 545.049,Z 240.218,A -85,B 0,C 180,E1 -3651.763,E2 -3651.763} C_VEL
LIN {X 0,Y 545.034,Z 240.208,A -85,B 0,C 180,E1 -3654.532,E2 -3654.532} C_VEL
LIN {X 0,Y 545.08,Z 240.213,A -85,B 0,C 180,E1 -3657.213,E2 -3657.213} C_VEL
LIN {X 0,Y 545.063,Z 240.216,A -85,B 0,C 180,E1 -3659.811,E2 -3659.811} C_VEL
LIN {X 0,Y 545.088,Z 240.21,A -85,B 0,C 180,E1 -3662.345,E2 -3662.345} C_VEL
LIN {X 0,Y 545.1,Z 240.316,A -85,B 0,C 180,E1 -3665.482,E2 -3665.482} C_VEL
LIN {X 0,Y 547.053,Z 249.178,A -85,B 0,C 180,E1 -3666.732,E2 -3666.732} C_VEL
LIN {X 0,Y 546.471,Z 272.888,A -85,B 0,C 180,E1 -3669.682,E2 -3669.682} C_VEL
LIN {X 0,Y 545.946,Z 294.905,A -85,B 0,C 180,E1 -3672.358,E2 -3672.358} C_VEL
LIN {X 0,Y 547.255,Z 302.683,A -85,B 0,C 180,E1 -3672.529,E2 -3672.529} C_VEL
LIN {X 0,Y 546.918,Z 423.051,A -85,B 0,C 180,E1 -3674.13,E2 -3674.13} C_VEL
LIN {X 0,Y 546.832,Z 438.882,A -85,B 0,C 180,E1 -3674.398,E2 -3674.398} C_VEL
LIN {X 0,Y 546.625,Z 452.835,A -85,B 0,C 180,E1 -3674.784,E2 -3674.784} C_VEL
LIN {X 0,Y 546.392,Z 466.798,A -85,B 0,C 180,E1 -3675.332,E2 -3675.332} C_VEL
LIN {X 0,Y 546.081,Z 480.443,A -85,B 0,C 180,E1 -3676.036,E2 -3676.036} C_VEL
LIN {X 0,Y 545.795,Z 493.372,A -85,B 0,C 180,E1 -3676.883,E2 -3676.883} C_VEL
LIN {X 0,Y 545.544,Z 504.955,A -85,B 0,C 180,E1 -3677.822,E2 -3677.822} C_VEL
LIN {X 0,Y 545.336,Z 515.394,A -85,B 0,C 180,E1 -3678.854,E2 -3678.854} C_VEL
LIN {X 0,Y 545.081,Z 524.824,A -85,B 0,C 180,E1 -3679.976,E2 -3679.976} C_VEL
LIN {X 0,Y 544.91,Z 533.804,A -85,B 0,C 180,E1 -3681.284,E2 -3681.284} C_VEL
LIN {X 0,Y 544.783,Z 541.055,A -85,B 0,C 180,E1 -3682.588,E2 -3682.588} C_VEL
LIN {X 0,Y 544.731,Z 547.569,A -85,B 0,C 180,E1 -3684.076,E2 -3684.076} C_VEL
LIN {X 0,Y 544.654,Z 552.444,A -85,B 0,C 180,E1 -3685.56,E2 -3685.56} C_VEL
LIN {X 0,Y 544.646,Z 555.833,A -85,B 0,C 180,E1 -3687.041,E2 -3687.041} C_VEL
LIN {X 0,Y 544.541,Z 557.835,A -85,B 0,C 180,E1 -3688.521,E2 -3688.521} C_VEL
LIN {X 0,Y 544.539,Z 558.5,A -85,B 0,C 180,E1 -3690,E2 -3690} C_VEL
LIN {X 0,Y 544.541,Z 557.836,A -85,B 0,C 180,E1 -3691.479,E2 -3691.479} C_VEL
LIN {X 0,Y 544.646,Z 555.836,A -85,B 0,C 180,E1 -3692.959,E2 -3692.959} C_VEL
LIN {X 0,Y 544.654,Z 552.447,A -85,B 0,C 180,E1 -3694.44,E2 -3694.44} C_VEL
LIN {X 0,Y 544.736,Z 547.568,A -85,B 0,C 180,E1 -3695.924,E2 -3695.924} C_VEL
LIN {X 0,Y 544.783,Z 541.054,A -85,B 0,C 180,E1 -3697.412,E2 -3697.412} C_VEL
LIN {X 0,Y 544.911,Z 533.804,A -85,B 0,C 180,E1 -3698.716,E2 -3698.716} C_VEL
LIN {X 0,Y 545.081,Z 524.822,A -85,B 0,C 180,E1 -3700.024,E2 -3700.024} C_VEL
LIN {X 0,Y 545.35,Z 515.394,A -85,B 0,C 180,E1 -3701.146,E2 -3701.146} C_VEL
LIN {X 0,Y 545.545,Z 504.952,A -85,B 0,C 180,E1 -3702.178,E2 -3702.178} C_VEL
LIN {X 0,Y 545.795,Z 493.372,A -85,B 0,C 180,E1 -3703.117,E2 -3703.117} C_VEL
LIN {X 0,Y 546.085,Z 480.444,A -85,B 0,C 180,E1 -3703.964,E2 -3703.964} C_VEL
LIN {X 0,Y 546.381,Z 466.784,A -85,B 0,C 180,E1 -3704.669,E2 -3704.669} C_VEL
LIN {X 0,Y 546.639,Z 453.514,A -85,B 0,C 180,E1 -3705.191,E2 -3705.191} C_VEL
LIN {X 0,Y 546.803,Z 439,A -85,B 0,C 180,E1 -3705.6,E2 -3705.6} C_VEL
LIN {X 0,Y 546.91,Z 422.96,A -85,B 0,C 180,E1 -3705.871,E2 -3705.871} C_VEL
LIN {X 0,Y 547.34,Z 303.183,A -85,B 0,C 180,E1 -3707.461,E2 -3707.461} C_VEL
LIN {X 0,Y 545.991,Z 295.34,A -85,B 0,C 180,E1 -3707.619,E2 -3707.619} C_VEL
LIN {X 0,Y 546.023,Z 290.315,A -85,B 0,C 180,E1 -3708.187,E2 -3708.187} C_VEL
LIN {X 0,Y 546.604,Z 266.564,A -85,B 0,C 180,E1 -3711.101,E2 -3711.101} C_VEL
LIN {X 0,Y 547.05,Z 249.178,A -85,B 0,C 180,E1 -3713.269,E2 -3713.269} C_VEL
LIN {X 0,Y 545.101,Z 240.317,A -85,B 0,C 180,E1 -3714.519,E2 -3714.519} C_VEL
LIN {X 0,Y 545.089,Z 240.21,A -85,B 0,C 180,E1 -3717.655,E2 -3717.655} C_VEL
LIN {X 0,Y 545.076,Z 240.214,A -85,B 0,C 180,E1 -3720.246,E2 -3720.246} C_VEL
LIN {X 0,Y 545.087,Z 240.209,A -85,B 0,C 180,E1 -3723.063,E2 -3723.063} C_VEL
LIN {X 0,Y 545.032,Z 240.212,A -85,B 0,C 180,E1 -3725.672,E2 -3725.672} C_VEL
LIN {X 0,Y 545.049,Z 240.215,A -85,B 0,C 180,E1 -3728.237,E2 -3728.237} C_VEL
LIN {X 0,Y 545.084,Z 240.206,A -85,B 0,C 180,E1 -3731.113,E2 -3731.113} C_VEL
LIN {X 0,Y 545.055,Z 240.217,A -85,B 0,C 180,E1 -3734.128,E2 -3734.128} C_VEL
LIN {X 0,Y 545.075,Z 240.209,A -85,B 0,C 180,E1 -3736.893,E2 -3736.893} C_VEL
LIN {X 0,Y 545.071,Z 240.21,A -85,B 0,C 180,E1 -3739.858,E2 -3739.858} C_VEL
LIN {X 0,Y 545.07,Z 240.206,A -85,B 0,C 180,E1 -3743.073,E2 -3743.073} C_VEL
LIN {X 0,Y 545.08,Z 240.208,A -85,B 0,C 180,E1 -3745.606,E2 -3745.606} C_VEL
LIN {X 0,Y 545.073,Z 240.211,A -85,B 0,C 180,E1 -3748.317,E2 -3748.317} C_VEL
LIN {X 0,Y 545.086,Z 240.203,A -85,B 0,C 180,E1 -3751.251,E2 -3751.251} C_VEL
LIN {X 0,Y 545.074,Z 240.217,A -85,B 0,C 180,E1 -3753.999,E2 -3753.999} C_VEL
LIN {X 0,Y 545.085,Z 240.209,A -85,B 0,C 180,E1 -3756.441,E2 -3756.441} C_VEL
LIN {X 0,Y 545.089,Z 240.211,A -85,B 0,C 180,E1 -3759.628,E2 -3759.628} C_VEL
LIN {X 0,Y 545.088,Z 240.206,A -85,B 0,C 180,E1 -3762.75,E2 -3762.75} C_VEL
LIN {X 0,Y 545.089,Z 240.215,A -85,B 0,C 180,E1 -3765.82,E2 -3765.82} C_VEL
LIN {X 0,Y 545.11,Z 240.202,A -85,B 0,C 180,E1 -3768.849,E2 -3768.849} C_VEL
LIN {X 0,Y 545.124,Z 240.206,A -85,B 0,C 180,E1 -3771.847,E2 -3771.847} C_VEL
LIN {X 0,Y 545.2,Z 240.193,A -85,B 0,C 180,E1 -3774.823,E2 -3774.823} C_VEL
LIN {X 0,Y 545.188,Z 240.199,A -85,B 0,C 180,E1 -3777.784,E2 -3777.784} C_VEL
LIN {X 0,Y 545.208,Z 240.192,A -85,B 0,C 180,E1 -3780.739,E2 -3780.739} C_VEL
LIN {X 0,Y 545.169,Z 240.196,A -85,B 0,C 180,E1 -3782.956,E2 -3782.956} C_VEL
LIN {X 0,Y 545.165,Z 240.198,A -85,B 0,C 180,E1 -3785.92,E2 -3785.92} C_VEL
LIN {X 0,Y 545.115,Z 240.205,A -85,B 0,C 180,E1 -3788.9,E2 -3788.9} C_VEL
LIN {X 0,Y 545.129,Z 240.202,A -85,B 0,C 180,E1 -3791.905,E2 -3791.905} C_VEL
LIN {X 0,Y 545.08,Z 240.211,A -85,B 0,C 180,E1 -3794.944,E2 -3794.944} C_VEL
LIN {X 0,Y 545.077,Z 240.208,A -85,B 0,C 180,E1 -3798.026,E2 -3798.026} C_VEL
LIN {X 0,Y 545.09,Z 240.205,A -85,B 0,C 180,E1 -3800.373,E2 -3800.373} C_VEL
LIN {X 0,Y 545.087,Z 240.209,A -85,B 0,C 180,E1 -3803.559,E2 -3803.559} C_VEL
LIN {X 0,Y 545.075,Z 240.208,A -85,B 0,C 180,E1 -3806.001,E2 -3806.001} C_VEL
LIN {X 0,Y 545.085,Z 240.208,A -85,B 0,C 180,E1 -3808.749,E2 -3808.749} C_VEL
LIN {X 0,Y 545.075,Z 240.21,A -85,B 0,C 180,E1 -3811.683,E2 -3811.683} C_VEL
LIN {X 0,Y 545.078,Z 240.209,A -85,B 0,C 180,E1 -3814.564,E2 -3814.564} C_VEL
LIN {X 0,Y 545.063,Z 240.216,A -85,B 0,C 180,E1 -3817.013,E2 -3817.013} C_VEL
LIN {X 0,Y 544.355,Z 240.302,A -85,B 0,C 180,E1 -3817.629,E2 -3817.629} C_VEL
LIN {X 0,Y 541.49,Z 240.66,A -85,B 0,C 180,E1 -3818.63,E2 -3818.63} C_VEL
LIN {X 0,Y 539.104,Z 240.951,A -85,B 0,C 180,E1 -3819.436,E2 -3819.436} C_VEL
LIN {X 0,Y 538.094,Z 241.074,A -85,B 0,C 180,E1 -3820.058,E2 -3820.058} C_VEL
LIN {X 0,Y 538.019,Z 241.084,A -85,B 0,C 180,E1 -3820.269,E2 -3820.269} C_VEL
LIN {X 0,Y 538.025,Z 241.091,A -85,B 0,C 180,E1 -3822.988,E2 -3822.988} C_VEL
LIN {X 0,Y 538.029,Z 241.087,A -85,B 0,C 180,E1 -3825.926,E2 -3825.926} C_VEL
LIN {X 0,Y 538.05,Z 241.086,A -85,B 0,C 180,E1 -3829.225,E2 -3829.225} C_VEL
LIN {X 0,Y 537.992,Z 241.083,A -85,B 0,C 180,E1 -3832.123,E2 -3832.123} C_VEL
LIN {X 0,Y 537.998,Z 241.091,A -85,B 0,C 180,E1 -3834.916,E2 -3834.916} C_VEL
LIN {X 0,Y 538.019,Z 241.09,A -85,B 0,C 180,E1 -3837.618,E2 -3837.618} C_VEL
LIN {X 0,Y 538.016,Z 241.093,A -85,B 0,C 180,E1 -3840.239,E2 -3840.239} C_VEL
LIN {X 0,Y 538.093,Z 241.25,A -85,B 0,C 180,E1 -3842.505,E2 -3842.505} C_VEL
LIN {X 0,Y 539.839,Z 250.213,A -85,B 0,C 180,E1 -3843.935,E2 -3843.935} C_VEL
LIN {X 0,Y 539.39,Z 269.882,A -85,B 0,C 180,E1 -3846.788,E2 -3846.788} C_VEL
LIN {X 0,Y 538.874,Z 290.309,A -85,B 0,C 180,E1 -3849.701,E2 -3849.701} C_VEL
LIN {X 0,Y 538.521,Z 310.428,A -85,B 0,C 180,E1 -3852.533,E2 -3852.533} C_VEL
LIN {X 0,Y 538.51,Z 315.601,A -85,B 0,C 180,E1 -3853.217,E2 -3853.217} C_VEL
LIN {X 0,Y 539.78,Z 325.034,A -85,B 0,C 180,E1 -3853.404,E2 -3853.404} C_VEL
LIN {X 0,Y 539.478,Z 424.394,A -85,B 0,C 180,E1 -3854.741,E2 -3854.741} C_VEL
LIN {X 0,Y 539.313,Z 436.588,A -85,B 0,C 180,E1 -3855.038,E2 -3855.038} C_VEL
LIN {X 0,Y 539.1,Z 449.648,A -85,B 0,C 180,E1 -3855.515,E2 -3855.515} C_VEL
LIN {X 0,Y 538.856,Z 460.309,A -85,B 0,C 180,E1 -3856.038,E2 -3856.038} C_VEL
LIN {X 0,Y 538.59,Z 471.023,A -85,B 0,C 180,E1 -3856.704,E2 -3856.704} C_VEL
LIN {X 0,Y 538.361,Z 481.941,A -85,B 0,C 180,E1 -3857.561,E2 -3857.561} C_VEL
LIN {X 0,Y 538.087,Z 492.162,A -85,B 0,C 180,E1 -3858.56,E2 -3858.56} C_VEL
LIN {X 0,Y 537.941,Z 501.16,A -85,B 0,C 180,E1 -3859.651,E2 -3859.651} C_VEL
LIN {X 0,Y 537.78,Z 508.683,A -85,B 0,C 180,E1 -3860.788,E2 -3860.788} C_VEL
LIN {X 0,Y 537.663,Z 515.631,A -85,B 0,C 180,E1 -3862.111,E2 -3862.111} C_VEL
LIN {X 0,Y 537.592,Z 521.085,A -85,B 0,C 180,E1 -3863.497,E2 -3863.497} C_VEL
LIN {X 0,Y 537.539,Z 524.651,A -85,B 0,C 180,E1 -3864.749,E2 -3864.749} C_VEL
LIN {X 0,Y 537.5,Z 526.226,A -85,B 0,C 180,E1 -3865.5,E2 -3865.5} C_VEL
LIN {X 0,Y 537.563,Z 527.388,A -85,B 0,C 180,E1 -3866.252,E2 -3866.252} C_VEL
LIN {X 0,Y 537.546,Z 528.114,A -85,B 0,C 180,E1 -3867.002,E2 -3867.002} C_VEL
LIN {X 0,Y 537.451,Z 528.427,A -85,B 0,C 180,E1 -3868.501,E2 -3868.501} C_VEL
LIN {X 0,Y 537.442,Z 528.009,A -85,B 0,C 180,E1 -3869.251,E2 -3869.251} C_VEL
LIN {X 0,Y 537.445,Z 527.162,A -85,B 0,C 180,E1 -3870,E2 -3870} C_VEL
LIN {X 0,Y 537.479,Z 524.28,A -85,B 0,C 180,E1 -3871.498,E2 -3871.498} C_VEL
LIN {X 0,Y 537.573,Z 520.987,A -85,B 0,C 180,E1 -3872.623,E2 -3872.623} C_VEL
LIN {X 0,Y 537.647,Z 516.647,A -85,B 0,C 180,E1 -3873.747,E2 -3873.747} C_VEL
LIN {X 0,Y 537.805,Z 511.133,A -85,B 0,C 180,E1 -3874.873,E2 -3874.873} C_VEL
LIN {X 0,Y 537.844,Z 504.272,A -85,B 0,C 180,E1 -3876,E2 -3876} C_VEL
LIN {X 0,Y 538.036,Z 496.011,A -85,B 0,C 180,E1 -3877.09,E2 -3877.09} C_VEL
LIN {X 0,Y 538.267,Z 486.914,A -85,B 0,C 180,E1 -3878.068,E2 -3878.068} C_VEL
LIN {X 0,Y 538.496,Z 477.29,A -85,B 0,C 180,E1 -3878.916,E2 -3878.916} C_VEL
LIN {X 0,Y 538.703,Z 466.764,A -85,B 0,C 180,E1 -3879.67,E2 -3879.67} C_VEL
LIN {X 0,Y 538.99,Z 455.007,A -85,B 0,C 180,E1 -3880.328,E2 -3880.328} C_VEL
LIN {X 0,Y 539.191,Z 442.811,A -85,B 0,C 180,E1 -3880.847,E2 -3880.847} C_VEL
LIN {X 0,Y 539.37,Z 430.296,A -85,B 0,C 180,E1 -3881.223,E2 -3881.223} C_VEL
LIN {X 0,Y 539.512,Z 417.341,A -85,B 0,C 180,E1 -3881.458,E2 -3881.458} C_VEL
LIN {X 0,Y 539.712,Z 323.421,A -85,B 0,C 180,E1 -3882.709,E2 -3882.709} C_VEL
LIN {X 0,Y 538.536,Z 315.706,A -85,B 0,C 180,E1 -3882.866,E2 -3882.866} C_VEL
LIN {X 0,Y 538.528,Z 311.576,A -85,B 0,C 180,E1 -3883.394,E2 -3883.394} C_VEL
LIN {X 0,Y 538.898,Z 291.06,A -85,B 0,C 180,E1 -3886.283,E2 -3886.283} C_VEL
LIN {X 0,Y 539.334,Z 271.906,A -85,B 0,C 180,E1 -3889.012,E2 -3889.012} C_VEL
LIN {X 0,Y 539.862,Z 251.401,A -85,B 0,C 180,E1 -3891.979,E2 -3891.979} C_VEL
LIN {X 0,Y 539.062,Z 245.866,A -85,B 0,C 180,E1 -3892.834,E2 -3892.834} C_VEL
LIN {X 0,Y 538.036,Z 241.16,A -85,B 0,C 180,E1 -3893.627,E2 -3893.627} C_VEL
LIN {X 0,Y 538.043,Z 241.078,A -85,B 0,C 180,E1 -3896.366,E2 -3896.366} C_VEL
LIN {X 0,Y 538.033,Z 241.09,A -85,B 0,C 180,E1 -3898.933,E2 -3898.933} C_VEL
LIN {X 0,Y 538.016,Z 241.09,A -85,B 0,C 180,E1 -3901.887,E2 -3901.887} C_VEL
LIN {X 0,Y 538.013,Z 241.085,A -85,B 0,C 180,E1 -3904.617,E2 -3904.617} C_VEL
LIN {X 0,Y 538.004,Z 241.097,A -85,B 0,C 180,E1 -3907.169,E2 -3907.169} C_VEL
LIN {X 0,Y 538.022,Z 241.089,A -85,B 0,C 180,E1 -3909.796,E2 -3909.796} C_VEL
LIN {X 0,Y 538.024,Z 241.089,A -85,B 0,C 180,E1 -3912.785,E2 -3912.785} C_VEL
LIN {X 0,Y 538.031,Z 241.09,A -85,B 0,C 180,E1 -3915.14,E2 -3915.14} C_VEL
LIN {X 0,Y 538.032,Z 241.085,A -85,B 0,C 180,E1 -3918.226,E2 -3918.226} C_VEL
LIN {X 0,Y 538.013,Z 241.093,A -85,B 0,C 180,E1 -3921.169,E2 -3921.169} C_VEL
LIN {X 0,Y 538.027,Z 241.086,A -85,B 0,C 180,E1 -3924.083,E2 -3924.083} C_VEL
LIN {X 0,Y 538.027,Z 241.085,A -85,B 0,C 180,E1 -3926.727,E2 -3926.727} C_VEL
LIN {X 0,Y 538.034,Z 241.087,A -85,B 0,C 180,E1 -3929.553,E2 -3929.553} C_VEL
LIN {X 0,Y 538.041,Z 241.082,A -85,B 0,C 180,E1 -3931.95,E2 -3931.95} C_VEL
LIN {X 0,Y 538.066,Z 241.085,A -85,B 0,C 180,E1 -3934.466,E2 -3934.466} C_VEL
LIN {X 0,Y 538.018,Z 241.096,A -85,B 0,C 180,E1 -3936.928,E2 -3936.928} C_VEL
LIN {X 0,Y 538.073,Z 241.08,A -85,B 0,C 180,E1 -3940.147,E2 -3940.147} C_VEL
LIN {X 0,Y 538.021,Z 241.088,A -85,B 0,C 180,E1 -3943.299,E2 -3943.299} C_VEL
LIN {X 0,Y 538.058,Z 241.08,A -85,B 0,C 180,E1 -3945.63,E2 -3945.63} C_VEL
LIN {X 0,Y 538.07,Z 241.087,A -85,B 0,C 180,E1 -3948.701,E2 -3948.701} C_VEL
LIN {X 0,Y 538.081,Z 241.079,A -85,B 0,C 180,E1 -3951.739,E2 -3951.739} C_VEL
LIN {X 0,Y 538.157,Z 241.073,A -85,B 0,C 180,E1 -3954.755,E2 -3954.755} C_VEL
LIN {X 0,Y 538.16,Z 241.07,A -85,B 0,C 180,E1 -3957.754,E2 -3957.754} C_VEL
LIN {X 0,Y 538.178,Z 241.07,A -85,B 0,C 180,E1 -3960.748,E2 -3960.748} C_VEL
LIN {X 0,Y 538.134,Z 241.074,A -85,B 0,C 180,E1 -3962.994,E2 -3962.994} C_VEL
LIN {X 0,Y 538.118,Z 241.076,A -85,B 0,C 180,E1 -3965.997,E2 -3965.997} C_VEL
LIN {X 0,Y 538.065,Z 241.082,A -85,B 0,C 180,E1 -3969.017,E2 -3969.017} C_VEL
LIN {X 0,Y 538.076,Z 241.083,A -85,B 0,C 180,E1 -3972.062,E2 -3972.062} C_VEL
LIN {X 0,Y 538.038,Z 241.083,A -85,B 0,C 180,E1 -3975.144,E2 -3975.144} C_VEL
LIN {X 0,Y 538.028,Z 241.094,A -85,B 0,C 180,E1 -3978.27,E2 -3978.27} C_VEL
LIN {X 0,Y 538.032,Z 241.086,A -85,B 0,C 180,E1 -3980.651,E2 -3980.651} C_VEL
LIN {X 0,Y 538.017,Z 241.094,A -85,B 0,C 180,E1 -3983.888,E2 -3983.888} C_VEL
LIN {X 0,Y 538.036,Z 241.089,A -85,B 0,C 180,E1 -3986.367,E2 -3986.367} C_VEL
LIN {X 0,Y 538.05,Z 241.08,A -85,B 0,C 180,E1 -3988.939,E2 -3988.939} C_VEL
LIN {X 0,Y 538.022,Z 241.09,A -85,B 0,C 180,E1 -3991.891,E2 -3991.891} C_VEL
LIN {X 0,Y 538.026,Z 241.087,A -85,B 0,C 180,E1 -3994.621,E2 -3994.621} C_VEL
LIN {X 0,Y 538.003,Z 241.084,A -85,B 0,C 180,E1 -3997.171,E2 -3997.171} C_VEL
LIN {X 0,Y 538.026,Z 241.096,A -85,B 0,C 180,E1 -3999.797,E2 -3999.797} C_VEL
LIN {X 0,Y 538.015,Z 241.086,A -85,B 0,C 180,E1 -4002.786,E2 -4002.786} C_VEL
LIN {X 0,Y 538.027,Z 241.087,A -85,B 0,C 180,E1 -4005.926,E2 -4005.926} C_VEL
LIN {X 0,Y 538.045,Z 241.078,A -85,B 0,C 180,E1 -4009.253,E2 -4009.253} C_VEL
LIN {X 0,Y 537.989,Z 241.092,A -85,B 0,C 180,E1 -4012.123,E2 -4012.123} C_VEL
LIN {X 0,Y 537.996,Z 241.086,A -85,B 0,C 180,E1 -4014.916,E2 -4014.916} C_VEL
LIN {X 0,Y 538.025,Z 241.088,A -85,B 0,C 180,E1 -4017.618,E2 -4017.618} C_VEL
LIN {X 0,Y 538.016,Z 241.09,A -85,B 0,C 180,E1 -4020.239,E2 -4020.239} C_VEL
LIN {X 0,Y 538.063,Z 241.086,A -85,B 0,C 180,E1 -4022.797,E2 -4022.797} C_VEL
LIN {X 0,Y 538.073,Z 241.259,A -85,B 0,C 180,E1 -4025.269,E2 -4025.269} C_VEL
LIN {X 0,Y 540.21,Z 250.775,A -85,B 0,C 180,E1 -4026.622,E2 -4026.622} C_VEL
LIN {X 0,Y 539.569,Z 274.621,A -85,B 0,C 180,E1 -4029.627,E2 -4029.627} C_VEL
LIN {X 0,Y 539.031,Z 295.162,A -85,B 0,C 180,E1 -4032.154,E2 -4032.154} C_VEL
LIN {X 0,Y 540.575,Z 305.612,A -85,B 0,C 180,E1 -4032.365,E2 -4032.365} C_VEL
LIN {X 0,Y 539.991,Z 433.652,A -85,B 0,C 180,E1 -4034.114,E2 -4034.114} C_VEL
LIN {X 0,Y 539.806,Z 447.847,A -85,B 0,C 180,E1 -4034.46,E2 -4034.46} C_VEL
LIN {X 0,Y 539.564,Z 461.634,A -85,B 0,C 180,E1 -4034.948,E2 -4034.948} C_VEL
LIN {X 0,Y 539.3,Z 474.757,A -85,B 0,C 180,E1 -4035.568,E2 -4035.568} C_VEL
LIN {X 0,Y 538.934,Z 487.45,A -85,B 0,C 180,E1 -4036.328,E2 -4036.328} C_VEL
LIN {X 0,Y 538.659,Z 499.019,A -85,B 0,C 180,E1 -4037.185,E2 -4037.185} C_VEL
LIN {X 0,Y 538.403,Z 510.014,A -85,B 0,C 180,E1 -4038.174,E2 -4038.174} C_VEL
LIN {X 0,Y 538.169,Z 520.151,A -85,B 0,C 180,E1 -4039.275,E2 -4039.275} C_VEL
LIN {X 0,Y 537.969,Z 528.822,A -85,B 0,C 180,E1 -4040.412,E2 -4040.412} C_VEL
LIN {X 0,Y 537.804,Z 537.11,A -85,B 0,C 180,E1 -4041.735,E2 -4041.735} C_VEL
LIN {X 0,Y 537.66,Z 542.864,A -85,B 0,C 180,E1 -4042.867,E2 -4042.867} C_VEL
LIN {X 0,Y 537.655,Z 548.961,A -85,B 0,C 180,E1 -4044.374,E2 -4044.374} C_VEL
LIN {X 0,Y 537.55,Z 552.444,A -85,B 0,C 180,E1 -4045.501,E2 -4045.501} C_VEL
LIN {X 0,Y 537.547,Z 555.832,A -85,B 0,C 180,E1 -4047.002,E2 -4047.002} C_VEL
LIN {X 0,Y 537.447,Z 557.835,A -85,B 0,C 180,E1 -4048.501,E2 -4048.501} C_VEL
LIN {X 0,Y 537.44,Z 558.5,A -85,B 0,C 180,E1 -4050,E2 -4050} C_VEL
LIN {X 0,Y 537.447,Z 557.837,A -85,B 0,C 180,E1 -4051.499,E2 -4051.499} C_VEL
LIN {X 0,Y 537.547,Z 555.836,A -85,B 0,C 180,E1 -4052.998,E2 -4052.998} C_VEL
LIN {X 0,Y 537.55,Z 552.447,A -85,B 0,C 180,E1 -4054.499,E2 -4054.499} C_VEL
LIN {X 0,Y 537.65,Z 547.567,A -85,B 0,C 180,E1 -4056.003,E2 -4056.003} C_VEL
LIN {X 0,Y 537.704,Z 541.054,A -85,B 0,C 180,E1 -4057.51,E2 -4057.51} C_VEL
LIN {X 0,Y 537.859,Z 533.765,A -85,B 0,C 180,E1 -4058.832,E2 -4058.832} C_VEL
LIN {X 0,Y 538.027,Z 524.688,A -85,B 0,C 180,E1 -4060.157,E2 -4060.157} C_VEL
LIN {X 0,Y 538.31,Z 515.151,A -85,B 0,C 180,E1 -4061.293,E2 -4061.293} C_VEL
LIN {X 0,Y 538.522,Z 504.568,A -85,B 0,C 180,E1 -4062.339,E2 -4062.339} C_VEL
LIN {X 0,Y 538.815,Z 492.871,A -85,B 0,C 180,E1 -4063.29,E2 -4063.29} C_VEL
LIN {X 0,Y 539.137,Z 479.862,A -85,B 0,C 180,E1 -4064.147,E2 -4064.147} C_VEL
LIN {X 0,Y 539.446,Z 466.087,A -85,B 0,C 180,E1 -4064.862,E2 -4064.862} C_VEL
LIN {X 0,Y 539.734,Z 452.08,A -85,B 0,C 180,E1 -4065.408,E2 -4065.408} C_VEL
LIN {X 0,Y 539.916,Z 437.925,A -85,B 0,C 180,E1 -4065.797,E2 -4065.797} C_VEL
LIN {X 0,Y 540.038,Z 422.648,A -85,B 0,C 180,E1 -4066.054,E2 -4066.054} C_VEL
LIN {X 0,Y 540.543,Z 304.158,A -85,B 0,C 180,E1 -4067.655,E2 -4067.655} C_VEL
LIN {X 0,Y 539.052,Z 295.197,A -85,B 0,C 180,E1 -4067.847,E2 -4067.847} C_VEL
LIN {X 0,Y 539.648,Z 271.318,A -85,B 0,C 180,E1 -4070.786,E2 -4070.786} C_VEL
LIN {X 0,Y 540.204,Z 250.772,A -85,B 0,C 180,E1 -4073.378,E2 -4073.378} C_VEL
LIN {X 0,Y 538.073,Z 241.189,A -85,B 0,C 180,E1 -4074.757,E2 -4074.757} C_VEL
LIN {X 0,Y 538.057,Z 241.087,A -85,B 0,C 180,E1 -4077.352,E2 -4077.352} C_VEL
LIN {X 0,Y 538.016,Z 241.089,A -85,B 0,C 180,E1 -4079.761,E2 -4079.761} C_VEL
LIN {X 0,Y 538.025,Z 241.086,A -85,B 0,C 180,E1 -4082.382,E2 -4082.382} C_VEL
LIN {X 0,Y 537.996,Z 241.089,A -85,B 0,C 180,E1 -4085.084,E2 -4085.084} C_VEL
LIN {X 0,Y 537.989,Z 241.089,A -85,B 0,C 180,E1 -4087.877,E2 -4087.877} C_VEL
LIN {X 0,Y 538.046,Z 241.086,A -85,B 0,C 180,E1 -4090.775,E2 -4090.775} C_VEL
LIN {X 0,Y 538.026,Z 241.092,A -85,B 0,C 180,E1 -4094.074,E2 -4094.074} C_VEL
LIN {X 0,Y 538.015,Z 241.088,A -85,B 0,C 180,E1 -4097.214,E2 -4097.214} C_VEL
LIN {X 0,Y 538.026,Z 241.093,A -85,B 0,C 180,E1 -4100.203,E2 -4100.203} C_VEL
LIN {X 0,Y 538.024,Z 241.084,A -85,B 0,C 180,E1 -4103.067,E2 -4103.067} C_VEL
LIN {X 0,Y 538.022,Z 241.09,A -85,B 0,C 180,E1 -4105.827,E2 -4105.827} C_VEL
LIN {X 0,Y 538.019,Z 241.087,A -85,B 0,C 180,E1 -4108.499,E2 -4108.499} C_VEL
LIN {X 0,Y 538.054,Z 241.078,A -85,B 0,C 180,E1 -4111.1,E2 -4111.1} C_VEL
LIN {X 0,Y 538.037,Z 241.089,A -85,B 0,C 180,E1 -4113.633,E2 -4113.633} C_VEL
LIN {X 0,Y 538.016,Z 241.094,A -85,B 0,C 180,E1 -4116.118,E2 -4116.118} C_VEL
LIN {X 0,Y 538.033,Z 241.086,A -85,B 0,C 180,E1 -4119.349,E2 -4119.349} C_VEL
LIN {X 0,Y 538.066,Z 241.081,A -85,B 0,C 180,E1 -4122.518,E2 -4122.518} C_VEL
LIN {X 0,Y 538.057,Z 241.089,A -85,B 0,C 180,E1 -4125.631,E2 -4125.631} C_VEL
LIN {X 0,Y 538.07,Z 241.079,A -85,B 0,C 180,E1 -4128.702,E2 -4128.702} C_VEL
LIN {X 0,Y 538.081,Z 241.085,A -85,B 0,C 180,E1 -4131.74,E2 -4131.74} C_VEL
LIN {X 0,Y 538.157,Z 241.07,A -85,B 0,C 180,E1 -4134.755,E2 -4134.755} C_VEL
LIN {X 0,Y 538.16,Z 241.075,A -85,B 0,C 180,E1 -4137.755,E2 -4137.755} C_VEL
LIN {X 0,Y 538.178,Z 241.068,A -85,B 0,C 180,E1 -4140.748,E2 -4140.748} C_VEL
LIN {X 0,Y 538.135,Z 241.072,A -85,B 0,C 180,E1 -4142.995,E2 -4142.995} C_VEL
LIN {X 0,Y 538.118,Z 241.075,A -85,B 0,C 180,E1 -4145.998,E2 -4145.998} C_VEL
LIN {X 0,Y 538.066,Z 241.085,A -85,B 0,C 180,E1 -4149.018,E2 -4149.018} C_VEL
LIN {X 0,Y 538.077,Z 241.079,A -85,B 0,C 180,E1 -4152.063,E2 -4152.063} C_VEL
LIN {X 0,Y 538.04,Z 241.091,A -85,B 0,C 180,E1 -4155.144,E2 -4155.144} C_VEL
LIN {X 0,Y 538.029,Z 241.086,A -85,B 0,C 180,E1 -4158.271,E2 -4158.271} C_VEL
LIN {X 0,Y 538.034,Z 241.085,A -85,B 0,C 180,E1 -4160.652,E2 -4160.652} C_VEL
LIN {X 0,Y 538.02,Z 241.086,A -85,B 0,C 180,E1 -4163.888,E2 -4163.888} C_VEL
LIN {X 0,Y 538.038,Z 241.086,A -85,B 0,C 180,E1 -4166.367,E2 -4166.367} C_VEL
LIN {X 0,Y 538.027,Z 241.088,A -85,B 0,C 180,E1 -4168.934,E2 -4168.934} C_VEL
LIN {X 0,Y 538.024,Z 241.087,A -85,B 0,C 180,E1 -4171.891,E2 -4171.891} C_VEL
LIN {X 0,Y 538.029,Z 241.088,A -85,B 0,C 180,E1 -4174.621,E2 -4174.621} C_VEL
LIN {X 0,Y 538.006,Z 241.095,A -85,B 0,C 180,E1 -4177.171,E2 -4177.171} C_VEL
LIN {X 0,Y 538.019,Z 241.084,A -85,B 0,C 180,E1 -4180.269,E2 -4180.269} C_VEL
LIN {X 0,Y 537.368,Z 241.173,A -85,B 0,C 180,E1 -4180.894,E2 -4180.894} C_VEL
LIN {X 0,Y 534.512,Z 241.528,A -85,B 0,C 180,E1 -4181.909,E2 -4181.909} C_VEL
LIN {X 0,Y 532.085,Z 241.834,A -85,B 0,C 180,E1 -4182.726,E2 -4182.726} C_VEL
LIN {X 0,Y 531.038,Z 241.957,A -85,B 0,C 180,E1 -4183.357,E2 -4183.357} C_VEL
LIN {X 0,Y 530.951,Z 241.966,A -85,B 0,C 180,E1 -4183.571,E2 -4183.571} C_VEL
LIN {X 0,Y 530.967,Z 241.972,A -85,B 0,C 180,E1 -4186.507,E2 -4186.507} C_VEL
LIN {X 0,Y 530.989,Z 241.969,A -85,B 0,C 180,E1 -4188.977,E2 -4188.977} C_VEL
LIN {X 0,Y 530.957,Z 241.957,A -85,B 0,C 180,E1 -4191.53,E2 -4191.53} C_VEL
LIN {X 0,Y 530.955,Z 241.974,A -85,B 0,C 180,E1 -4194.381,E2 -4194.381} C_VEL
LIN {X 0,Y 530.968,Z 241.971,A -85,B 0,C 180,E1 -4197.134,E2 -4197.134} C_VEL
LIN {X 0,Y 530.963,Z 241.968,A -85,B 0,C 180,E1 -4199.803,E2 -4199.803} C_VEL
LIN {X 0,Y 531.056,Z 242.126,A -85,B 0,C 180,E1 -4202.274,E2 -4202.274} C_VEL
LIN {X 0,Y 532.986,Z 252.008,A -85,B 0,C 180,E1 -4203.877,E2 -4203.877} C_VEL
LIN {X 0,Y 532.479,Z 271.061,A -85,B 0,C 180,E1 -4206.675,E2 -4206.675} C_VEL
LIN {X 0,Y 531.938,Z 290.496,A -85,B 0,C 180,E1 -4209.481,E2 -4209.481} C_VEL
LIN {X 0,Y 531.586,Z 310.233,A -85,B 0,C 180,E1 -4212.298,E2 -4212.298} C_VEL
LIN {X 0,Y 531.521,Z 315.338,A -85,B 0,C 180,E1 -4212.99,E2 -4212.99} C_VEL
LIN {X 0,Y 532.964,Z 325.787,A -85,B 0,C 180,E1 -4213.202,E2 -4213.202} C_VEL
LIN {X 0,Y 532.659,Z 424.274,A -85,B 0,C 180,E1 -4214.536,E2 -4214.536} C_VEL
LIN {X 0,Y 532.468,Z 436.721,A -85,B 0,C 180,E1 -4214.841,E2 -4214.841} C_VEL
LIN {X 0,Y 532.236,Z 449.78,A -85,B 0,C 180,E1 -4215.324,E2 -4215.324} C_VEL
LIN {X 0,Y 531.961,Z 460.439,A -85,B 0,C 180,E1 -4215.853,E2 -4215.853} C_VEL
LIN {X 0,Y 531.67,Z 471.146,A -85,B 0,C 180,E1 -4216.528,E2 -4216.528} C_VEL
LIN {X 0,Y 531.42,Z 482.063,A -85,B 0,C 180,E1 -4217.396,E2 -4217.396} C_VEL
LIN {X 0,Y 531.13,Z 491.211,A -85,B 0,C 180,E1 -4218.29,E2 -4218.29} C_VEL
LIN {X 0,Y 530.942,Z 499.841,A -85,B 0,C 180,E1 -4219.321,E2 -4219.321} C_VEL
LIN {X 0,Y 530.732,Z 507.698,A -85,B 0,C 180,E1 -4220.472,E2 -4220.472} C_VEL
LIN {X 0,Y 530.608,Z 513.967,A -85,B 0,C 180,E1 -4221.622,E2 -4221.622} C_VEL
LIN {X 0,Y 530.567,Z 518.952,A -85,B 0,C 180,E1 -4222.771,E2 -4222.771} C_VEL
LIN {X 0,Y 530.471,Z 522.818,A -85,B 0,C 180,E1 -4223.916,E2 -4223.916} C_VEL
LIN {X 0,Y 530.463,Z 524.808,A -85,B 0,C 180,E1 -4224.679,E2 -4224.679} C_VEL
LIN {X 0,Y 530.406,Z 526.387,A -85,B 0,C 180,E1 -4225.44,E2 -4225.44} C_VEL
LIN {X 0,Y 530.482,Z 527.559,A -85,B 0,C 180,E1 -4226.202,E2 -4226.202} C_VEL
LIN {X 0,Y 530.41,Z 528.652,A -85,B 0,C 180,E1 -4227.722,E2 -4227.722} C_VEL
LIN {X 0,Y 530.345,Z 528.229,A -85,B 0,C 180,E1 -4229.241,E2 -4229.241} C_VEL
LIN {X 0,Y 530.35,Z 527.404,A -85,B 0,C 180,E1 -4230,E2 -4230} C_VEL
LIN {X 0,Y 530.39,Z 524.556,A -85,B 0,C 180,E1 -4231.519,E2 -4231.519} C_VEL
LIN {X 0,Y 530.494,Z 521.305,A -85,B 0,C 180,E1 -4232.658,E2 -4232.658} C_VEL
LIN {X 0,Y 530.57,Z 517.009,A -85,B 0,C 180,E1 -4233.797,E2 -4233.797} C_VEL
LIN {X 0,Y 530.747,Z 511.544,A -85,B 0,C 180,E1 -4234.937,E2 -4234.937} C_VEL
LIN {X 0,Y 530.807,Z 504.747,A -85,B 0,C 180,E1 -4236.08,E2 -4236.08} C_VEL
LIN {X 0,Y 531.026,Z 496.258,A -85,B 0,C 180,E1 -4237.222,E2 -4237.222} C_VEL
LIN {X 0,Y 531.287,Z 487.564,A -85,B 0,C 180,E1 -4238.175,E2 -4238.175} C_VEL
LIN {X 0,Y 531.533,Z 478.048,A -85,B 0,C 180,E1 -4239.033,E2 -4239.033} C_VEL
LIN {X 0,Y 531.758,Z 467.67,A -85,B 0,C 180,E1 -4239.797,E2 -4239.797} C_VEL
LIN {X 0,Y 532.086,Z 456.209,A -85,B 0,C 180,E1 -4240.464,E2 -4240.464} C_VEL
LIN {X 0,Y 532.307,Z 444.35,A -85,B 0,C 180,E1 -4240.989,E2 -4240.989} C_VEL
LIN {X 0,Y 532.495,Z 431.515,A -85,B 0,C 180,E1 -4241.394,E2 -4241.394} C_VEL
LIN {X 0,Y 532.674,Z 417.799,A -85,B 0,C 180,E1 -4241.655,E2 -4241.655} C_VEL
LIN {X 0,Y 532.936,Z 324.465,A -85,B 0,C 180,E1 -4242.906,E2 -4242.906} C_VEL
LIN {X 0,Y 531.56,Z 315.543,A -85,B 0,C 180,E1 -4243.086,E2 -4243.086} C_VEL
LIN {X 0,Y 531.615,Z 307.665,A -85,B 0,C 180,E1 -4244.156,E2 -4244.156} C_VEL
LIN {X 0,Y 532.064,Z 287.13,A -85,B 0,C 180,E1 -4247.091,E2 -4247.091} C_VEL
LIN {X 0,Y 532.592,Z 266.613,A -85,B 0,C 180,E1 -4250.065,E2 -4250.065} C_VEL
LIN {X 0,Y 532.968,Z 251.571,A -85,B 0,C 180,E1 -4252.278,E2 -4252.278} C_VEL
LIN {X 0,Y 531.015,Z 242.104,A -85,B 0,C 180,E1 -4253.808,E2 -4253.808} C_VEL
LIN {X 0,Y 531.002,Z 241.955,A -85,B 0,C 180,E1 -4256.743,E2 -4256.743} C_VEL
LIN {X 0,Y 530.984,Z 241.966,A -85,B 0,C 180,E1 -4259.322,E2 -4259.322} C_VEL
LIN {X 0,Y 530.972,Z 241.966,A -85,B 0,C 180,E1 -4262.1,E2 -4262.1} C_VEL
LIN {X 0,Y 530.971,Z 241.963,A -85,B 0,C 180,E1 -4264.85,E2 -4264.85} C_VEL
LIN {X 0,Y 530.965,Z 241.971,A -85,B 0,C 180,E1 -4267.507,E2 -4267.507} C_VEL
LIN {X 0,Y 530.981,Z 241.964,A -85,B 0,C 180,E1 -4270.432,E2 -4270.432} C_VEL
LIN {X 0,Y 530.971,Z 241.973,A -85,B 0,C 180,E1 -4273.281,E2 -4273.281} C_VEL
LIN {X 0,Y 530.983,Z 241.966,A -85,B 0,C 180,E1 -4275.62,E2 -4275.62} C_VEL
LIN {X 0,Y 530.994,Z 241.964,A -85,B 0,C 180,E1 -4278.564,E2 -4278.564} C_VEL
LIN {X 0,Y 530.957,Z 241.97,A -85,B 0,C 180,E1 -4281.529,E2 -4281.529} C_VEL
LIN {X 0,Y 530.979,Z 241.965,A -85,B 0,C 180,E1 -4284.381,E2 -4284.381} C_VEL
LIN {X 0,Y 530.969,Z 241.968,A -85,B 0,C 180,E1 -4287.133,E2 -4287.133} C_VEL
LIN {X 0,Y 530.982,Z 241.964,A -85,B 0,C 180,E1 -4289.803,E2 -4289.803} C_VEL
LIN {X 0,Y 531.011,Z 241.961,A -85,B 0,C 180,E1 -4292.466,E2 -4292.466} C_VEL
LIN {X 0,Y 531.001,Z 241.967,A -85,B 0,C 180,E1 -4294.942,E2 -4294.942} C_VEL
LIN {X 0,Y 530.966,Z 241.968,A -85,B 0,C 180,E1 -4298.246,E2 -4298.246} C_VEL
LIN {X 0,Y 530.992,Z 241.968,A -85,B 0,C 180,E1 -4300.677,E2 -4300.677} C_VEL
LIN {X 0,Y 530.987,Z 241.967,A -85,B 0,C 180,E1 -4303.071,E2 -4303.071} C_VEL
LIN {X 0,Y 531.013,Z 241.959,A -85,B 0,C 180,E1 -4305.435,E2 -4305.435} C_VEL
LIN {X 0,Y 531.03,Z 241.966,A -85,B 0,C 180,E1 -4308.549,E2 -4308.549} C_VEL
LIN {X 0,Y 531.05,Z 241.954,A -85,B 0,C 180,E1 -4311.629,E2 -4311.629} C_VEL
LIN {X 0,Y 531.116,Z 241.951,A -85,B 0,C 180,E1 -4314.685,E2 -4314.685} C_VEL
LIN {X 0,Y 531.132,Z 241.945,A -85,B 0,C 180,E1 -4317.725,E2 -4317.725} C_VEL
LIN {X 0,Y 531.148,Z 241.946,A -85,B 0,C 180,E1 -4320.758,E2 -4320.758} C_VEL
LIN {X 0,Y 531.101,Z 241.95,A -85,B 0,C 180,E1 -4323.034,E2 -4323.034} C_VEL
LIN {X 0,Y 531.077,Z 241.954,A -85,B 0,C 180,E1 -4326.077,E2 -4326.077} C_VEL
LIN {X 0,Y 531.025,Z 241.958,A -85,B 0,C 180,E1 -4329.138,E2 -4329.138} C_VEL
LIN {X 0,Y 531.033,Z 241.963,A -85,B 0,C 180,E1 -4332.225,E2 -4332.225} C_VEL
LIN {X 0,Y 530.989,Z 241.961,A -85,B 0,C 180,E1 -4335.35,E2 -4335.35} C_VEL
LIN {X 0,Y 531.009,Z 241.963,A -85,B 0,C 180,E1 -4337.722,E2 -4337.722} C_VEL
LIN {X 0,Y 530.992,Z 241.961,A -85,B 0,C 180,E1 -4340.938,E2 -4340.938} C_VEL
LIN {X 0,Y 530.973,Z 241.97,A -85,B 0,C 180,E1 -4344.225,E2 -4344.225} C_VEL
LIN {X 0,Y 531,Z 241.962,A -85,B 0,C 180,E1 -4346.744,E2 -4346.744} C_VEL
LIN {X 0,Y 530.994,Z 241.96,A -85,B 0,C 180,E1 -4349.322,E2 -4349.322} C_VEL
LIN {X 0,Y 530.974,Z 241.972,A -85,B 0,C 180,E1 -4352.103,E2 -4352.103} C_VEL
LIN {X 0,Y 530.983,Z 241.963,A -85,B 0,C 180,E1 -4354.855,E2 -4354.855} C_VEL
LIN {X 0,Y 530.961,Z 241.964,A -85,B 0,C 180,E1 -4357.508,E2 -4357.508} C_VEL
LIN {X 0,Y 530.98,Z 241.965,A -85,B 0,C 180,E1 -4360.433,E2 -4360.433} C_VEL
LIN {X 0,Y 530.959,Z 241.967,A -85,B 0,C 180,E1 -4363.282,E2 -4363.282} C_VEL
LIN {X 0,Y 530.984,Z 241.97,A -85,B 0,C 180,E1 -4365.621,E2 -4365.621} C_VEL
LIN {X 0,Y 530.994,Z 241.952,A -85,B 0,C 180,E1 -4368.565,E2 -4368.565} C_VEL
LIN {X 0,Y 530.954,Z 241.975,A -85,B 0,C 180,E1 -4371.53,E2 -4371.53} C_VEL
LIN {X 0,Y 530.951,Z 241.962,A -85,B 0,C 180,E1 -4374.381,E2 -4374.381} C_VEL
LIN {X 0,Y 530.968,Z 241.971,A -85,B 0,C 180,E1 -4377.134,E2 -4377.134} C_VEL
LIN {X 0,Y 530.968,Z 241.972,A -85,B 0,C 180,E1 -4379.804,E2 -4379.804} C_VEL
LIN {X 0,Y 531.014,Z 241.964,A -85,B 0,C 180,E1 -4382.467,E2 -4382.467} C_VEL
LIN {X 0,Y 531.07,Z 242.111,A -85,B 0,C 180,E1 -4385.025,E2 -4385.025} C_VEL
LIN {X 0,Y 533.357,Z 252.378,A -85,B 0,C 180,E1 -4386.51,E2 -4386.51} C_VEL
LIN {X 0,Y 532.652,Z 275.957,A -85,B 0,C 180,E1 -4389.521,E2 -4389.521} C_VEL
LIN {X 0,Y 532.123,Z 295.467,A -85,B 0,C 180,E1 -4391.945,E2 -4391.945} C_VEL
LIN {X 0,Y 533.747,Z 305.518,A -85,B 0,C 180,E1 -4392.153,E2 -4392.153} C_VEL
LIN {X 0,Y 533.106,Z 433.416,A -85,B 0,C 180,E1 -4393.928,E2 -4393.928} C_VEL
LIN {X 0,Y 532.898,Z 447.989,A -85,B 0,C 180,E1 -4394.289,E2 -4394.289} C_VEL
LIN {X 0,Y 532.63,Z 462.011,A -85,B 0,C 180,E1 -4394.797,E2 -4394.797} C_VEL
LIN {X 0,Y 532.365,Z 474.128,A -85,B 0,C 180,E1 -4395.376,E2 -4395.376} C_VEL
LIN {X 0,Y 531.981,Z 486.916,A -85,B 0,C 180,E1 -4396.146,E2 -4396.146} C_VEL
LIN {X 0,Y 531.68,Z 498.555,A -85,B 0,C 180,E1 -4397.014,E2 -4397.014} C_VEL
LIN {X 0,Y 531.363,Z 510.06,A -85,B 0,C 180,E1 -4398.06,E2 -4398.06} C_VEL
LIN {X 0,Y 531.147,Z 519.79,A -85,B 0,C 180,E1 -4399.132,E2 -4399.132} C_VEL
LIN {X 0,Y 530.894,Z 528.497,A -85,B 0,C 180,E1 -4400.283,E2 -4400.283} C_VEL
LIN {X 0,Y 530.736,Z 536.829,A -85,B 0,C 180,E1 -4401.625,E2 -4401.625} C_VEL
LIN {X 0,Y 530.585,Z 542.636,A -85,B 0,C 180,E1 -4402.771,E2 -4402.771} C_VEL
LIN {X 0,Y 530.564,Z 548.811,A -85,B 0,C 180,E1 -4404.299,E2 -4404.299} C_VEL
LIN {X 0,Y 530.447,Z 552.325,A -85,B 0,C 180,E1 -4405.441,E2 -4405.441} C_VEL
LIN {X 0,Y 530.452,Z 555.748,A -85,B 0,C 180,E1 -4406.962,E2 -4406.962} C_VEL
LIN {X 0,Y 530.357,Z 557.769,A -85,B 0,C 180,E1 -4408.481,E2 -4408.481} C_VEL
LIN {X 0,Y 530.341,Z 558.439,A -85,B 0,C 180,E1 -4410,E2 -4410} C_VEL
LIN {X 0,Y 530.357,Z 557.77,A -85,B 0,C 180,E1 -4411.519,E2 -4411.519} C_VEL
LIN {X 0,Y 530.452,Z 555.752,A -85,B 0,C 180,E1 -4413.038,E2 -4413.038} C_VEL
LIN {X 0,Y 530.447,Z 552.329,A -85,B 0,C 180,E1 -4414.56,E2 -4414.56} C_VEL
LIN {X 0,Y 530.546,Z 547.4,A -85,B 0,C 180,E1 -4416.083,E2 -4416.083} C_VEL
LIN {X 0,Y 530.64,Z 540.812,A -85,B 0,C 180,E1 -4417.611,E2 -4417.611} C_VEL
LIN {X 0,Y 530.794,Z 533.468,A -85,B 0,C 180,E1 -4418.95,E2 -4418.95} C_VEL
LIN {X 0,Y 531.001,Z 524.344,A -85,B 0,C 180,E1 -4420.293,E2 -4420.293} C_VEL
LIN {X 0,Y 531.262,Z 514.763,A -85,B 0,C 180,E1 -4421.445,E2 -4421.445} C_VEL
LIN {X 0,Y 531.527,Z 504.132,A -85,B 0,C 180,E1 -4422.504,E2 -4422.504} C_VEL
LIN {X 0,Y 531.835,Z 492.37,A -85,B 0,C 180,E1 -4423.468,E2 -4423.468} C_VEL
LIN {X 0,Y 532.162,Z 480.877,A -85,B 0,C 180,E1 -4424.239,E2 -4424.239} C_VEL
LIN {X 0,Y 532.479,Z 467.398,A -85,B 0,C 180,E1 -4424.963,E2 -4424.963} C_VEL
LIN {X 0,Y 532.788,Z 453.936,A -85,B 0,C 180,E1 -4425.516,E2 -4425.516} C_VEL
LIN {X 0,Y 533.008,Z 439.517,A -85,B 0,C 180,E1 -4425.942,E2 -4425.942} C_VEL
LIN {X 0,Y 533.161,Z 424.14,A -85,B 0,C 180,E1 -4426.217,E2 -4426.217} C_VEL
LIN {X 0,Y 533.705,Z 304.794,A -85,B 0,C 180,E1 -4427.858,E2 -4427.858} C_VEL
LIN {X 0,Y 532.164,Z 295.437,A -85,B 0,C 180,E1 -4428.057,E2 -4428.057} C_VEL
LIN {X 0,Y 532.818,Z 269.741,A -85,B 0,C 180,E1 -4431.268,E2 -4431.268} C_VEL
LIN {X 0,Y 533.347,Z 252.371,A -85,B 0,C 180,E1 -4433.491,E2 -4433.491} C_VEL
LIN {X 0,Y 531.058,Z 242.082,A -85,B 0,C 180,E1 -4434.989,E2 -4434.989} C_VEL
LIN {X 0,Y 531.015,Z 241.964,A -85,B 0,C 180,E1 -4437.595,E2 -4437.595} C_VEL
LIN {X 0,Y 530.973,Z 241.969,A -85,B 0,C 180,E1 -4440.645,E2 -4440.645} C_VEL
LIN {X 0,Y 530.985,Z 241.965,A -85,B 0,C 180,E1 -4443.772,E2 -4443.772} C_VEL
LIN {X 0,Y 530.952,Z 241.964,A -85,B 0,C 180,E1 -4446.558,E2 -4446.558} C_VEL
LIN {X 0,Y 530.983,Z 241.965,A -85,B 0,C 180,E1 -4449.443,E2 -4449.443} C_VEL
LIN {X 0,Y 530.979,Z 241.972,A -85,B 0,C 180,E1 -4452.456,E2 -4452.456} C_VEL
LIN {X 0,Y 530.982,Z 241.964,A -85,B 0,C 180,E1 -4455.621,E2 -4455.621} C_VEL
LIN {X 0,Y 530.996,Z 241.962,A -85,B 0,C 180,E1 -4458.565,E2 -4458.565} C_VEL
LIN {X 0,Y 530.955,Z 241.969,A -85,B 0,C 180,E1 -4461.529,E2 -4461.529} C_VEL
LIN {X 0,Y 530.977,Z 241.967,A -85,B 0,C 180,E1 -4464.382,E2 -4464.382} C_VEL
LIN {X 0,Y 530.967,Z 241.966,A -85,B 0,C 180,E1 -4467.133,E2 -4467.133} C_VEL
LIN {X 0,Y 530.981,Z 241.965,A -85,B 0,C 180,E1 -4469.804,E2 -4469.804} C_VEL
LIN {X 0,Y 531.01,Z 241.963,A -85,B 0,C 180,E1 -4472.466,E2 -4472.466} C_VEL
LIN {X 0,Y 530.999,Z 241.961,A -85,B 0,C 180,E1 -4474.942,E2 -4474.942} C_VEL
LIN {X 0,Y 530.965,Z 241.969,A -85,B 0,C 180,E1 -4478.247,E2 -4478.247} C_VEL
LIN {X 0,Y 530.99,Z 241.963,A -85,B 0,C 180,E1 -4480.677,E2 -4480.677} C_VEL
LIN {X 0,Y 530.986,Z 241.963,A -85,B 0,C 180,E1 -4483.071,E2 -4483.071} C_VEL
LIN {X 0,Y 531.012,Z 241.963,A -85,B 0,C 180,E1 -4485.436,E2 -4485.436} C_VEL
LIN {X 0,Y 531.029,Z 241.956,A -85,B 0,C 180,E1 -4488.55,E2 -4488.55} C_VEL
LIN {X 0,Y 531.05,Z 241.963,A -85,B 0,C 180,E1 -4491.63,E2 -4491.63} C_VEL
LIN {X 0,Y 531.116,Z 241.947,A -85,B 0,C 180,E1 -4494.685,E2 -4494.685} C_VEL
LIN {X 0,Y 531.132,Z 241.951,A -85,B 0,C 180,E1 -4497.725,E2 -4497.725} C_VEL
LIN {X 0,Y 531.148,Z 241.943,A -85,B 0,C 180,E1 -4500.758,E2 -4500.758} C_VEL
LIN {X 0,Y 531.102,Z 241.949,A -85,B 0,C 180,E1 -4503.034,E2 -4503.034} C_VEL
LIN {X 0,Y 531.078,Z 241.951,A -85,B 0,C 180,E1 -4506.077,E2 -4506.077} C_VEL
LIN {X 0,Y 531.026,Z 241.963,A -85,B 0,C 180,E1 -4509.139,E2 -4509.139} C_VEL
LIN {X 0,Y 531.035,Z 241.956,A -85,B 0,C 180,E1 -4512.225,E2 -4512.225} C_VEL
LIN {X 0,Y 530.99,Z 241.968,A -85,B 0,C 180,E1 -4515.35,E2 -4515.35} C_VEL
LIN {X 0,Y 531.011,Z 241.963,A -85,B 0,C 180,E1 -4517.723,E2 -4517.723} C_VEL
LIN {X 0,Y 530.995,Z 241.965,A -85,B 0,C 180,E1 -4520.938,E2 -4520.938} C_VEL
LIN {X 0,Y 530.975,Z 241.963,A -85,B 0,C 180,E1 -4524.225,E2 -4524.225} C_VEL
LIN {X 0,Y 531.001,Z 241.966,A -85,B 0,C 180,E1 -4526.744,E2 -4526.744} C_VEL
LIN {X 0,Y 530.978,Z 241.965,A -85,B 0,C 180,E1 -4529.323,E2 -4529.323} C_VEL
LIN {X 0,Y 530.977,Z 241.965,A -85,B 0,C 180,E1 -4532.104,E2 -4532.104} C_VEL
LIN {X 0,Y 530.986,Z 241.966,A -85,B 0,C 180,E1 -4534.855,E2 -4534.855} C_VEL
LIN {X 0,Y 530.965,Z 241.968,A -85,B 0,C 180,E1 -4537.508,E2 -4537.508} C_VEL
LIN {X 0,Y 530.982,Z 241.962,A -85,B 0,C 180,E1 -4540.433,E2 -4540.433} C_VEL
LIN {X 0,Y 530.96,Z 241.967,A -85,B 0,C 180,E1 -4543.282,E2 -4543.282} C_VEL
LIN {X 0,Y 530.951,Z 241.966,A -85,B 0,C 180,E1 -4543.571,E2 -4543.571} C_VEL
LIN {X 0,Y 530.283,Z 242.05,A -85,B 0,C 180,E1 -4544.204,E2 -4544.204} C_VEL
LIN {X 0,Y 527.442,Z 242.411,A -85,B 0,C 180,E1 -4545.233,E2 -4545.233} C_VEL
LIN {X 0,Y 525.041,Z 242.714,A -85,B 0,C 180,E1 -4546.062,E2 -4546.062} C_VEL
LIN {X 0,Y 524.008,Z 242.84,A -85,B 0,C 180,E1 -4546.702,E2 -4546.702} C_VEL
LIN {X 0,Y 523.923,Z 242.847,A -85,B 0,C 180,E1 -4546.918,E2 -4546.918} C_VEL
LIN {X 0,Y 523.949,Z 242.841,A -85,B 0,C 180,E1 -4549.921,E2 -4549.921} C_VEL
LIN {X 0,Y 523.908,Z 242.847,A -85,B 0,C 180,E1 -4552.869,E2 -4552.869} C_VEL
LIN {X 0,Y 523.921,Z 242.839,A -85,B 0,C 180,E1 -4555.71,E2 -4555.71} C_VEL
LIN {X 0,Y 523.921,Z 242.847,A -85,B 0,C 180,E1 -4558.456,E2 -4558.456} C_VEL
LIN {X 0,Y 523.933,Z 242.842,A -85,B 0,C 180,E1 -4561.125,E2 -4561.125} C_VEL
LIN {X 0,Y 524.02,Z 243.047,A -85,B 0,C 180,E1 -4562.048,E2 -4562.048} C_VEL
LIN {X 0,Y 525.925,Z 252.133,A -85,B 0,C 180,E1 -4563.552,E2 -4563.552} C_VEL
LIN {X 0,Y 526.05,Z 256.803,A -85,B 0,C 180,E1 -4564.266,E2 -4564.266} C_VEL
LIN {X 0,Y 525.407,Z 278.519,A -85,B 0,C 180,E1 -4567.483,E2 -4567.483} C_VEL
LIN {X 0,Y 524.8,Z 300.258,A -85,B 0,C 180,E1 -4570.644,E2 -4570.644} C_VEL
LIN {X 0,Y 524.533,Z 315.082,A -85,B 0,C 180,E1 -4572.756,E2 -4572.756} C_VEL
LIN {X 0,Y 525.807,Z 323.077,A -85,B 0,C 180,E1 -4572.936,E2 -4572.936} C_VEL
LIN {X 0,Y 526.195,Z 329.662,A -85,B 0,C 180,E1 -4573.037,E2 -4573.037} C_VEL
LIN {X 0,Y 525.844,Z 424.506,A -85,B 0,C 180,E1 -4574.332,E2 -4574.332} C_VEL
LIN {X 0,Y 525.626,Z 436.887,A -85,B 0,C 180,E1 -4574.639,E2 -4574.639} C_VEL
LIN {X 0,Y 525.381,Z 449.948,A -85,B 0,C 180,E1 -4575.128,E2 -4575.128} C_VEL
LIN {X 0,Y 525.037,Z 462.323,A -85,B 0,C 180,E1 -4575.762,E2 -4575.762} C_VEL
LIN {X 0,Y 524.675,Z 473.926,A -85,B 0,C 180,E1 -4576.542,E2 -4576.542} C_VEL
LIN {X 0,Y 524.376,Z 484.348,A -85,B 0,C 180,E1 -4577.421,E2 -4577.421} C_VEL
LIN {X 0,Y 524.055,Z 493.741,A -85,B 0,C 180,E1 -4578.395,E2 -4578.395} C_VEL
LIN {X 0,Y 523.856,Z 502.779,A -85,B 0,C 180,E1 -4579.565,E2 -4579.565} C_VEL
LIN {X 0,Y 523.679,Z 510.063,A -85,B 0,C 180,E1 -4580.733,E2 -4580.733} C_VEL
LIN {X 0,Y 523.526,Z 515.902,A -85,B 0,C 180,E1 -4581.897,E2 -4581.897} C_VEL
LIN {X 0,Y 523.484,Z 520.508,A -85,B 0,C 180,E1 -4583.06,E2 -4583.06} C_VEL
LIN {X 0,Y 523.391,Z 522.97,A -85,B 0,C 180,E1 -4583.833,E2 -4583.833} C_VEL
LIN {X 0,Y 523.389,Z 524.962,A -85,B 0,C 180,E1 -4584.607,E2 -4584.607} C_VEL
LIN {X 0,Y 523.314,Z 526.546,A -85,B 0,C 180,E1 -4585.378,E2 -4585.378} C_VEL
LIN {X 0,Y 523.402,Z 527.729,A -85,B 0,C 180,E1 -4586.15,E2 -4586.15} C_VEL
LIN {X 0,Y 523.334,Z 528.845,A -85,B 0,C 180,E1 -4587.691,E2 -4587.691} C_VEL
LIN {X 0,Y 523.251,Z 528.446,A -85,B 0,C 180,E1 -4589.23,E2 -4589.23} C_VEL
LIN {X 0,Y 523.254,Z 527.646,A -85,B 0,C 180,E1 -4590,E2 -4590} C_VEL
LIN {X 0,Y 523.304,Z 524.833,A -85,B 0,C 180,E1 -4591.539,E2 -4591.539} C_VEL
LIN {X 0,Y 523.418,Z 521.619,A -85,B 0,C 180,E1 -4592.694,E2 -4592.694} C_VEL
LIN {X 0,Y 523.498,Z 517.367,A -85,B 0,C 180,E1 -4593.849,E2 -4593.849} C_VEL
LIN {X 0,Y 523.69,Z 511.953,A -85,B 0,C 180,E1 -4595.004,E2 -4595.004} C_VEL
LIN {X 0,Y 523.774,Z 505.221,A -85,B 0,C 180,E1 -4596.162,E2 -4596.162} C_VEL
LIN {X 0,Y 524.006,Z 497.156,A -85,B 0,C 180,E1 -4597.281,E2 -4597.281} C_VEL
LIN {X 0,Y 524.315,Z 488.238,A -85,B 0,C 180,E1 -4598.285,E2 -4598.285} C_VEL
LIN {X 0,Y 524.63,Z 477.681,A -85,B 0,C 180,E1 -4599.25,E2 -4599.25} C_VEL
LIN {X 0,Y 524.916,Z 467.188,A -85,B 0,C 180,E1 -4600.023,E2 -4600.023} C_VEL
LIN {X 0,Y 525.223,Z 455.489,A -85,B 0,C 180,E1 -4600.699,E2 -4600.699} C_VEL
LIN {X 0,Y 525.493,Z 443.351,A -85,B 0,C 180,E1 -4601.23,E2 -4601.23} C_VEL
LIN {X 0,Y 525.703,Z 430.008,A -85,B 0,C 180,E1 -4601.641,E2 -4601.641} C_VEL
LIN {X 0,Y 525.856,Z 414.743,A -85,B 0,C 180,E1 -4601.907,E2 -4601.907} C_VEL
LIN {X 0,Y 526.114,Z 325.117,A -85,B 0,C 180,E1 -4603.116,E2 -4603.116} C_VEL
LIN {X 0,Y 524.592,Z 315.384,A -85,B 0,C 180,E1 -4603.312,E2 -4603.312} C_VEL
LIN {X 0,Y 524.654,Z 307.864,A -85,B 0,C 180,E1 -4604.348,E2 -4604.348} C_VEL
LIN {X 0,Y 525.192,Z 285.943,A -85,B 0,C 180,E1 -4607.523,E2 -4607.523} C_VEL
LIN {X 0,Y 525.75,Z 265.585,A -85,B 0,C 180,E1 -4610.516,E2 -4610.516} C_VEL
LIN {X 0,Y 526.124,Z 253.398,A -85,B 0,C 180,E1 -4612.33,E2 -4612.33} C_VEL
LIN {X 0,Y 523.949,Z 242.924,A -85,B 0,C 180,E1 -4614.059,E2 -4614.059} C_VEL
LIN {X 0,Y 523.976,Z 242.823,A -85,B 0,C 180,E1 -4616.271,E2 -4616.271} C_VEL
LIN {X 0,Y 523.957,Z 242.84,A -85,B 0,C 180,E1 -4619.323,E2 -4619.323} C_VEL
LIN {X 0,Y 523.938,Z 242.841,A -85,B 0,C 180,E1 -4622.449,E2 -4622.449} C_VEL
LIN {X 0,Y 523.921,Z 242.846,A -85,B 0,C 180,E1 -4625.226,E2 -4625.226} C_VEL
LIN {X 0,Y 523.914,Z 242.844,A -85,B 0,C 180,E1 -4628.101,E2 -4628.101} C_VEL
LIN {X 0,Y 523.961,Z 242.843,A -85,B 0,C 180,E1 -4631.31,E2 -4631.31} C_VEL
LIN {X 0,Y 523.955,Z 242.84,A -85,B 0,C 180,E1 -4634.69,E2 -4634.69} C_VEL
LIN {X 0,Y 523.951,Z 242.84,A -85,B 0,C 180,E1 -4637.88,E2 -4637.88} C_VEL
LIN {X 0,Y 523.921,Z 242.843,A -85,B 0,C 180,E1 -4640.915,E2 -4640.915} C_VEL
LIN {X 0,Y 523.925,Z 242.843,A -85,B 0,C 180,E1 -4643.827,E2 -4643.827} C_VEL
LIN {X 0,Y 523.939,Z 242.837,A -85,B 0,C 180,E1 -4646.635,E2 -4646.635} C_VEL
LIN {X 0,Y 523.96,Z 242.842,A -85,B 0,C 180,E1 -4649.355,E2 -4649.355} C_VEL
LIN {X 0,Y 523.974,Z 242.836,A -85,B 0,C 180,E1 -4652.28,E2 -4652.28} C_VEL
LIN {X 0,Y 523.948,Z 242.845,A -85,B 0,C 180,E1 -4654.581,E2 -4654.581} C_VEL
LIN {X 0,Y 523.911,Z 242.85,A -85,B 0,C 180,E1 -4657.106,E2 -4657.106} C_VEL
LIN {X 0,Y 523.973,Z 242.835,A -85,B 0,C 180,E1 -4659.865,E2 -4659.865} C_VEL
LIN {X 0,Y 523.965,Z 242.845,A -85,B 0,C 180,E1 -4662.837,E2 -4662.837} C_VEL
LIN {X 0,Y 523.97,Z 242.837,A -85,B 0,C 180,E1 -4665.235,E2 -4665.235} C_VEL
LIN {X 0,Y 524.005,Z 242.838,A -85,B 0,C 180,E1 -4668.394,E2 -4668.394} C_VEL
LIN {X 0,Y 523.998,Z 242.833,A -85,B 0,C 180,E1 -4671.516,E2 -4671.516} C_VEL
LIN {X 0,Y 524.077,Z 242.828,A -85,B 0,C 180,E1 -4674.613,E2 -4674.613} C_VEL
LIN {X 0,Y 524.105,Z 242.821,A -85,B 0,C 180,E1 -4677.694,E2 -4677.694} C_VEL
LIN {X 0,Y 524.118,Z 242.821,A -85,B 0,C 180,E1 -4680.768,E2 -4680.768} C_VEL
LIN {X 0,Y 524.067,Z 242.826,A -85,B 0,C 180,E1 -4683.075,E2 -4683.075} C_VEL
LIN {X 0,Y 524.039,Z 242.832,A -85,B 0,C 180,E1 -4686.159,E2 -4686.159} C_VEL
LIN {X 0,Y 523.993,Z 242.834,A -85,B 0,C 180,E1 -4689.262,E2 -4689.262} C_VEL
LIN {X 0,Y 523.995,Z 242.833,A -85,B 0,C 180,E1 -4691.739,E2 -4691.739} C_VEL
LIN {X 0,Y 523.985,Z 242.834,A -85,B 0,C 180,E1 -4695.052,E2 -4695.052} C_VEL
LIN {X 0,Y 523.957,Z 242.844,A -85,B 0,C 180,E1 -4697.969,E2 -4697.969} C_VEL
LIN {X 0,Y 523.964,Z 242.841,A -85,B 0,C 180,E1 -4700.41,E2 -4700.41} C_VEL
LIN {X 0,Y 523.91,Z 242.845,A -85,B 0,C 180,E1 -4702.893,E2 -4702.893} C_VEL
LIN {X 0,Y 523.946,Z 242.84,A -85,B 0,C 180,E1 -4705.419,E2 -4705.419} C_VEL
LIN {X 0,Y 523.964,Z 242.844,A -85,B 0,C 180,E1 -4707.999,E2 -4707.999} C_VEL
LIN {X 0,Y 523.946,Z 242.834,A -85,B 0,C 180,E1 -4710.857,E2 -4710.857} C_VEL
LIN {X 0,Y 523.955,Z 242.845,A -85,B 0,C 180,E1 -4713.735,E2 -4713.735} C_VEL
LIN {X 0,Y 523.917,Z 242.839,A -85,B 0,C 180,E1 -4716.405,E2 -4716.405} C_VEL
LIN {X 0,Y 523.919,Z 242.845,A -85,B 0,C 180,E1 -4719.085,E2 -4719.085} C_VEL
LIN {X 0,Y 523.952,Z 242.841,A -85,B 0,C 180,E1 -4722.119,E2 -4722.119} C_VEL
LIN {X 0,Y 523.952,Z 242.843,A -85,B 0,C 180,E1 -4725.309,E2 -4725.309} C_VEL
LIN {X 0,Y 523.955,Z 242.828,A -85,B 0,C 180,E1 -4728.69,E2 -4728.69} C_VEL
LIN {X 0,Y 523.914,Z 242.846,A -85,B 0,C 180,E1 -4731.081,E2 -4731.081} C_VEL
LIN {X 0,Y 523.897,Z 242.842,A -85,B 0,C 180,E1 -4733.826,E2 -4733.826} C_VEL
LIN {X 0,Y 523.94,Z 242.843,A -85,B 0,C 180,E1 -4736.636,E2 -4736.636} C_VEL
LIN {X 0,Y 523.954,Z 242.841,A -85,B 0,C 180,E1 -4739.356,E2 -4739.356} C_VEL
LIN {X 0,Y 523.978,Z 242.841,A -85,B 0,C 180,E1 -4742.282,E2 -4742.282} C_VEL
LIN {X 0,Y 524.021,Z 243.029,A -85,B 0,C 180,E1 -4744.798,E2 -4744.798} C_VEL
LIN {X 0,Y 526.491,Z 253.971,A -85,B 0,C 180,E1 -4746.393,E2 -4746.393} C_VEL
LIN {X 0,Y 525.837,Z 275.372,A -85,B 0,C 180,E1 -4749.166,E2 -4749.166} C_VEL
LIN {X 0,Y 525.21,Z 295.583,A -85,B 0,C 180,E1 -4751.719,E2 -4751.719} C_VEL
LIN {X 0,Y 526.956,Z 306.713,A -85,B 0,C 180,E1 -4751.953,E2 -4751.953} C_VEL
LIN {X 0,Y 526.212,Z 433.076,A -85,B 0,C 180,E1 -4753.735,E2 -4753.735} C_VEL
LIN {X 0,Y 525.996,Z 447.415,A -85,B 0,C 180,E1 -4754.09,E2 -4754.09} C_VEL
LIN {X 0,Y 525.711,Z 461.246,A -85,B 0,C 180,E1 -4754.592,E2 -4754.592} C_VEL
LIN {X 0,Y 525.37,Z 475.28,A -85,B 0,C 180,E1 -4755.276,E2 -4755.276} C_VEL
LIN {X 0,Y 524.997,Z 487.824,A -85,B 0,C 180,E1 -4756.057,E2 -4756.057} C_VEL
LIN {X 0,Y 524.658,Z 499.278,A -85,B 0,C 180,E1 -4756.936,E2 -4756.936} C_VEL
LIN {X 0,Y 524.335,Z 510.413,A -85,B 0,C 180,E1 -4757.973,E2 -4757.973} C_VEL
LIN {X 0,Y 524.063,Z 521.002,A -85,B 0,C 180,E1 -4759.179,E2 -4759.179} C_VEL
LIN {X 0,Y 523.809,Z 529.479,A -85,B 0,C 180,E1 -4760.345,E2 -4760.345} C_VEL
LIN {X 0,Y 523.634,Z 537.565,A -85,B 0,C 180,E1 -4761.704,E2 -4761.704} C_VEL
LIN {X 0,Y 523.494,Z 544.068,A -85,B 0,C 180,E1 -4763.06,E2 -4763.06} C_VEL
LIN {X 0,Y 523.448,Z 549.825,A -85,B 0,C 180,E1 -4764.607,E2 -4764.607} C_VEL
LIN {X 0,Y 523.418,Z 554,A -85,B 0,C 180,E1 -4766.151,E2 -4766.151} C_VEL
LIN {X 0,Y 523.333,Z 556.724,A -85,B 0,C 180,E1 -4767.691,E2 -4767.691} C_VEL
LIN {X 0,Y 523.247,Z 558.072,A -85,B 0,C 180,E1 -4769.23,E2 -4769.23} C_VEL
LIN {X 0,Y 523.247,Z 558.072,A -85,B 0,C 180,E1 -4770.77,E2 -4770.77} C_VEL
LIN {X 0,Y 523.333,Z 556.726,A -85,B 0,C 180,E1 -4772.309,E2 -4772.309} C_VEL
LIN {X 0,Y 523.418,Z 554.006,A -85,B 0,C 180,E1 -4773.849,E2 -4773.849} C_VEL
LIN {X 0,Y 523.449,Z 549.829,A -85,B 0,C 180,E1 -4775.393,E2 -4775.393} C_VEL
LIN {X 0,Y 523.494,Z 544.07,A -85,B 0,C 180,E1 -4776.94,E2 -4776.94} C_VEL
LIN {X 0,Y 523.634,Z 537.567,A -85,B 0,C 180,E1 -4778.296,E2 -4778.296} C_VEL
LIN {X 0,Y 523.807,Z 529.475,A -85,B 0,C 180,E1 -4779.655,E2 -4779.655} C_VEL
LIN {X 0,Y 524.072,Z 520.997,A -85,B 0,C 180,E1 -4780.821,E2 -4780.821} C_VEL
LIN {X 0,Y 524.339,Z 511.477,A -85,B 0,C 180,E1 -4781.914,E2 -4781.914} C_VEL
LIN {X 0,Y 524.634,Z 500.439,A -85,B 0,C 180,E1 -4782.966,E2 -4782.966} C_VEL
LIN {X 0,Y 524.935,Z 489.24,A -85,B 0,C 180,E1 -4783.846,E2 -4783.846} C_VEL
